gfCNCPoint2[13248] = {X 390.9830, Y 62.2246, Z -3.0000, A 0.000, B 0.000, C 0.000 }
gfCNCPoint2[13249] = {X 390.3072, Y 62.7207, Z -3.0000, A 0.000, B 0.000, C 0.000 }
gfCNCPoint2[13250] = {X 389.5499, Y 63.0803, Z -3.0000, A 0.000, B 0.000, C 0.000 }
gfCNCPoint2[13251] = {X 388.7383, Y 63.2905, Z -3.0000, A 0.000, B 0.000, C 0.000 }
gfCNCPoint2[13252] = {X 388.7383, Y 83.9247, Z -3.0000, A 0.000, B 0.000, C 0.000 }
gfCNCPoint2[13253] = {X 388.7363, Y 84.6149, Z -3.0000, A 0.000, B 0.000, C 0.000 }
gfCNCPoint2[13254] = {X 388.6762, Y 86.2799, Z -3.0000, A 0.000, B 0.000, C 0.000 }
gfCNCPoint2[13255] = {X 388.4710, Y 87.9334, Z -3.0000, A 0.000, B 0.000, C 0.000 }
gfCNCPoint2[13256] = {X 388.1223, Y 89.5626, Z -3.0000, A 0.000, B 0.000, C 0.000 }
gfCNCPoint2[13257] = {X 387.5865, Y 91.1607, Z -3.0000, A 0.000, B 0.000, C 0.000 }
gfCNCPoint2[13258] = {X 386.8319, Y 92.6679, Z -3.0000, A 0.000, B 0.000, C 0.000 }
gfCNCPoint2[13259] = {X 385.8732, Y 94.0543, Z -3.0000, A 0.000, B 0.000, C 0.000 }
gfCNCPoint2[13260] = {X 384.7295, Y 95.2924, Z -3.0000, A 0.000, B 0.000, C 0.000 }
gfCNCPoint2[13261] = {X 383.5014, Y 96.3480, Z -3.0000, A 0.000, B 0.000, C 0.000 }
gfCNCPoint2[13262] = {X 382.1865, Y 97.2935, Z -3.0000, A 0.000, B 0.000, C 0.000 }
gfCNCPoint2[13263] = {X 382.4496, Y 97.6950, Z -3.0000, A 0.000, B 0.000, C 0.000 }
gfCNCPoint2[13264] = {X 391.5259, Y 97.6950, Z -3.0000, A 0.000, B 0.000, C 0.000 }
gfCNCPoint2[13265] = {X 391.5259, Y 97.0659, Z -3.0000, A 0.000, B 0.000, C 0.000 }
gfCNCPoint2[13266] = {X 391.6192, Y 96.1166, Z -3.0000, A 0.000, B 0.000, C 0.000 }
gfCNCPoint2[13267] = {X 391.8953, Y 95.2035, Z -3.0000, A 0.000, B 0.000, C 0.000 }
gfCNCPoint2[13268] = {X 392.3439, Y 94.3615, Z -3.0000, A 0.000, B 0.000, C 0.000 }
gfCNCPoint2[13269] = {X 392.9476, Y 93.6229, Z -3.0000, A 0.000, B 0.000, C 0.000 }
gfCNCPoint2[13270] = {X 393.6835, Y 93.0159, Z -3.0000, A 0.000, B 0.000, C 0.000 }
gfCNCPoint2[13271] = {X 394.5234, Y 92.5637, Z -3.0000, A 0.000, B 0.000, C 0.000 }
gfCNCPoint2[13272] = {X 395.4353, Y 92.2834, Z -3.0000, A 0.000, B 0.000, C 0.000 }
gfCNCPoint2[13273] = {X 396.3843, Y 92.1860, Z -3.0000, A 0.000, B 0.000, C 0.000 }
gfCNCPoint2[13274] = {X 397.3061, Y 92.1465, Z -3.0000, A 0.000, B 0.000, C 0.000 }
gfCNCPoint2[13275] = {X 398.2246, Y 92.0592, Z -3.0000, A 0.000, B 0.000, C 0.000 }
gfCNCPoint2[13276] = {X 398.7527, Y 91.9311, Z -3.0000, A 0.000, B 0.000, C 0.000 }
gfCNCPoint2[13277] = {X 399.2389, Y 91.6885, Z -3.0000, A 0.000, B 0.000, C 0.000 }
gfCNCPoint2[13278] = {X 426.8276, Y 74.0193, Z -3.0000, A 0.000, B 0.000, C 0.000 }
gfCNCPoint2[13279] = {X 403.5508, Y 64.8864, Z -3.0000, A 0.000, B 0.000, C 0.000 }
gfCNCPoint2[13280] = {X 401.9168, Y 64.3451, Z -3.0000, A 0.000, B 0.000, C 0.000 }
gfCNCPoint2[13281] = {X 400.2332, Y 63.9861, Z -3.0000, A 0.000, B 0.000, C 0.000 }
gfCNCPoint2[13282] = {X 398.5205, Y 63.8139, Z -3.0000, A 0.000, B 0.000, C 0.000 }
gfCNCPoint2[13283] = {X 397.5547, Y 63.7099, Z -3.0000, A 0.000, B 0.000, C 0.000 }
gfCNCPoint2[13284] = {X 396.6287, Y 63.4166, Z -3.0000, A 0.000, B 0.000, C 0.000 }
gfCNCPoint2[13285] = {X 395.7791, Y 62.9458, Z -3.0000, A 0.000, B 0.000, C 0.000 }
gfCNCPoint2[13286] = {X 395.0396, Y 62.3160, Z -3.0000, A 0.000, B 0.000, C 0.000 }
gfCNCPoint2[13287] = {X 394.4659, Y 61.5933, Z -3.0000, A 0.000, B 0.000, C 0.000 }
gfCNCPoint2[13288] = {X 394.0385, Y 60.7756, Z -3.0000, A 0.000, B 0.000, C 0.000 }
gfCNCPoint2[13289] = {X 393.7727, Y 59.8921, Z -3.0000, A 0.000, B 0.000, C 0.000 }
gfCNCPoint2[13290] = {X 393.6779, Y 58.9744, Z -3.0000, A 0.000, B 0.000, C 0.000 }
gfCNCPoint2[13291] = {X 393.6777, Y 58.0000, Z -3.0000, A 0.000, B 0.000, C 0.000 }
gfCNCPoint2[13292] = {X 393.7668, Y 57.0718, Z -3.0000, A 0.000, B 0.000, C 0.000 }
gfCNCPoint2[13293] = {X 394.0309, Y 56.1774, Z -3.0000, A 0.000, B 0.000, C 0.000 }
gfCNCPoint2[13294] = {X 394.4602, Y 55.3496, Z -3.0000, A 0.000, B 0.000, C 0.000 }
gfCNCPoint2[13295] = {X 395.0391, Y 54.6186, Z -3.0000, A 0.000, B 0.000, C 0.000 }
gfCNCPoint2[13296] = {X 395.7864, Y 53.9833, Z -3.0000, A 0.000, B 0.000, C 0.000 }
gfCNCPoint2[13297] = {X 396.6455, Y 53.5102, Z -3.0000, A 0.000, B 0.000, C 0.000 }
gfCNCPoint2[13298] = {X 397.5819, Y 53.2186, Z -3.0000, A 0.000, B 0.000, C 0.000 }
gfCNCPoint2[13299] = {X 398.5577, Y 53.1200, Z -3.0000, A 0.000, B 0.000, C 0.000 }
gfCNCPoint2[13300] = {X 419.4886, Y 53.1200, Z -3.0000, A 0.000, B 0.000, C 0.000 }
gfCNCPoint2[13301] = {X 420.5534, Y 53.2376, Z -3.0000, A 0.000, B 0.000, C 0.000 }
gfCNCPoint2[13302] = {X 421.5670, Y 53.5847, Z -3.0000, A 0.000, B 0.000, C 0.000 }
gfCNCPoint2[13303] = {X 422.4803, Y 54.1446, Z -3.0000, A 0.000, B 0.000, C 0.000 }
gfCNCPoint2[13304] = {X 423.2495, Y 54.8903, Z -3.0000, A 0.000, B 0.000, C 0.000 }
gfCNCPoint2[13305] = {X 423.8374, Y 55.7859, Z -3.0000, A 0.000, B 0.000, C 0.000 }
gfCNCPoint2[13306] = {X 424.2157, Y 56.7881, Z -3.0000, A 0.000, B 0.000, C 0.000 }
gfCNCPoint2[13307] = {X 424.3663, Y 57.8488, Z -3.0000, A 0.000, B 0.000, C 0.000 }
gfCNCPoint2[13308] = {X 429.8190, Y 59.9739, Z -3.0000, A 0.000, B 0.000, C 0.000 }
gfCNCPoint2[13309] = {X 457.3006, Y 70.8772, Z -3.0000, A 0.000, B 0.000, C 0.000 }
gfCNCPoint2[13310] = {X 457.2996, Y 63.6742, Z -3.0000, A 0.000, B 0.000, C 0.000 }
gfCNCPoint2[13311] = {X 456.2913, Y 63.3059, Z -3.0000, A 0.000, B 0.000, C 0.000 }
gfCNCPoint2[13312] = {X 455.3879, Y 62.7260, Z -3.0000, A 0.000, B 0.000, C 0.000 }
gfCNCPoint2[13313] = {X 454.6331, Y 61.9627, Z -3.0000, A 0.000, B 0.000, C 0.000 }
gfCNCPoint2[13314] = {X 454.0635, Y 61.0528, Z -3.0000, A 0.000, B 0.000, C 0.000 }
gfCNCPoint2[13315] = {X 453.7067, Y 60.0403, Z -3.0000, A 0.000, B 0.000, C 0.000 }
gfCNCPoint2[13316] = {X 453.5798, Y 58.9744, Z -3.0000, A 0.000, B 0.000, C 0.000 }
gfCNCPoint2[13317] = {X 453.5796, Y 58.0000, Z -3.0000, A 0.000, B 0.000, C 0.000 }
gfCNCPoint2[13318] = {X 453.6734, Y 57.0480, Z -3.0000, A 0.000, B 0.000, C 0.000 }
gfCNCPoint2[13319] = {X 453.9511, Y 56.1325, Z -3.0000, A 0.000, B 0.000, C 0.000 }
gfCNCPoint2[13320] = {X 454.4020, Y 55.2888, Z -3.0000, A 0.000, B 0.000, C 0.000 }
gfCNCPoint2[13321] = {X 455.0089, Y 54.5493, Z -3.0000, A 0.000, B 0.000, C 0.000 }
gfCNCPoint2[13322] = {X 455.7484, Y 53.9424, Z -3.0000, A 0.000, B 0.000, C 0.000 }
gfCNCPoint2[13323] = {X 456.5921, Y 53.4915, Z -3.0000, A 0.000, B 0.000, C 0.000 }
gfCNCPoint2[13324] = {X 457.5076, Y 53.2138, Z -3.0000, A 0.000, B 0.000, C 0.000 }
gfCNCPoint2[13325] = {X 458.4596, Y 53.1200, Z -3.0000, A 0.000, B 0.000, C 0.000 }
gfCNCPoint2[13326] = {X 475.0000, Y 53.1200, Z -3.0000, A 0.000, B 0.000, C 0.000 }
gfCNCPoint2[13327] = {X 475.9520, Y 53.2138, Z -3.0000, A 0.000, B 0.000, C 0.000 }
gfCNCPoint2[13328] = {X 476.8675, Y 53.4915, Z -3.0000, A 0.000, B 0.000, C 0.000 }
gfCNCPoint2[13329] = {X 477.7112, Y 53.9424, Z -3.0000, A 0.000, B 0.000, C 0.000 }
gfCNCPoint2[13330] = {X 478.4507, Y 54.5493, Z -3.0000, A 0.000, B 0.000, C 0.000 }
gfCNCPoint2[13331] = {X 479.0576, Y 55.2888, Z -3.0000, A 0.000, B 0.000, C 0.000 }
gfCNCPoint2[13332] = {X 479.5085, Y 56.1325, Z -3.0000, A 0.000, B 0.000, C 0.000 }
gfCNCPoint2[13333] = {X 479.7862, Y 57.0480, Z -3.0000, A 0.000, B 0.000, C 0.000 }
gfCNCPoint2[13334] = {X 479.8800, Y 58.0000, Z -3.0000, A 0.000, B 0.000, C 0.000 }
gfCNCPoint2[13335] = {X 479.8798, Y 58.9744, Z -3.0000, A 0.000, B 0.000, C 0.000 }
gfCNCPoint2[13336] = {X 479.7529, Y 60.0404, Z -3.0000, A 0.000, B 0.000, C 0.000 }
gfCNCPoint2[13337] = {X 479.3960, Y 61.0529, Z -3.0000, A 0.000, B 0.000, C 0.000 }
gfCNCPoint2[13338] = {X 478.8264, Y 61.9628, Z -3.0000, A 0.000, B 0.000, C 0.000 }
gfCNCPoint2[13339] = {X 478.0716, Y 62.7261, Z -3.0000, A 0.000, B 0.000, C 0.000 }
gfCNCPoint2[13340] = {X 477.1681, Y 63.3060, Z -3.0000, A 0.000, B 0.000, C 0.000 }
gfCNCPoint2[13341] = {X 476.1597, Y 63.6743, Z -3.0000, A 0.000, B 0.000, C 0.000 }
gfCNCPoint2[13342] = {X 476.1601, Y 92.3320, Z -3.0000, A 0.000, B 0.000, C 0.000 }
gfCNCPoint2[13343] = {X 476.3629, Y 92.3914, Z -3.0000, A 0.000, B 0.000, C 0.000 }
gfCNCPoint2[13344] = {X 476.5640, Y 92.4558, Z -3.0000, A 0.000, B 0.000, C 0.000 }
gfCNCPoint2[13345] = {X 477.4819, Y 92.8728, Z -3.0000, A 0.000, B 0.000, C 0.000 }
gfCNCPoint2[13346] = {X 478.2938, Y 93.4704, Z -3.0000, A 0.000, B 0.000, C 0.000 }
gfCNCPoint2[13347] = {X 478.9647, Y 94.2227, Z -3.0000, A 0.000, B 0.000, C 0.000 }
gfCNCPoint2[13348] = {X 479.4658, Y 95.0975, Z -3.0000, A 0.000, B 0.000, C 0.000 }
gfCNCPoint2[13349] = {X 479.7753, Y 96.0569, Z -3.0000, A 0.000, B 0.000, C 0.000 }
gfCNCPoint2[13350] = {X 479.8800, Y 97.0595, Z -3.0000, A 0.000, B 0.000, C 0.000 }
gfCNCPoint2[13351] = {X 479.8800, Y 97.6950, Z -3.0000, A 0.000, B 0.000, C 0.000 }
gfCNCPoint2[13352] = {X 479.4000, Y 97.6950, Z -3.0000, A 0.000, B 0.000, C 0.000 }
gfCNCPoint2[13353] = {X 479.4000, Y 98.0000, Z -3.0000, A 0.000, B 0.000, C 0.000 }
gfCNCPoint2[13354] = {X 479.2897, Y 98.9791, Z -3.0000, A 0.000, B 0.000, C 0.000 }
gfCNCPoint2[13355] = {X 478.9643, Y 99.9091, Z -3.0000, A 0.000, B 0.000, C 0.000 }
gfCNCPoint2[13356] = {X 478.4401, Y 100.7434, Z -3.0000, A 0.000, B 0.000, C 0.000 }
gfCNCPoint2[13357] = {X 477.7434, Y 101.4401, Z -3.0000, A 0.000, B 0.000, C 0.000 }
gfCNCPoint2[13358] = {X 476.9091, Y 101.9643, Z -3.0000, A 0.000, B 0.000, C 0.000 }
gfCNCPoint2[13359] = {X 475.9791, Y 102.2897, Z -3.0000, A 0.000, B 0.000, C 0.000 }
gfCNCPoint2[13360] = {X 475.0000, Y 102.4000, Z -3.0000, A 0.000, B 0.000, C 0.000 }
gfCNCPoint2[13361] = {X 458.4596, Y 102.4000, Z -3.0000, A 0.000, B 0.000, C 0.000 }
gfCNCPoint2[13362] = {X 457.4805, Y 102.2897, Z -3.0000, A 0.000, B 0.000, C 0.000 }
gfCNCPoint2[13363] = {X 456.5505, Y 101.9643, Z -3.0000, A 0.000, B 0.000, C 0.000 }
gfCNCPoint2[13364] = {X 455.7162, Y 101.4401, Z -3.0000, A 0.000, B 0.000, C 0.000 }
gfCNCPoint2[13365] = {X 455.0195, Y 100.7434, Z -3.0000, A 0.000, B 0.000, C 0.000 }
gfCNCPoint2[13366] = {X 454.4953, Y 99.9091, Z -3.0000, A 0.000, B 0.000, C 0.000 }
gfCNCPoint2[13367] = {X 454.1699, Y 98.9791, Z -3.0000, A 0.000, B 0.000, C 0.000 }
gfCNCPoint2[13368] = {X 454.0596, Y 98.0000, Z -3.0000, A 0.000, B 0.000, C 0.000 }
gfCNCPoint2[13369] = {X 454.0596, Y 97.0659, Z -3.0000, A 0.000, B 0.000, C 0.000 }
gfCNCPoint2[13370] = {X 454.1492, Y 96.1826, Z -3.0000, A 0.000, B 0.000, C 0.000 }
gfCNCPoint2[13371] = {X 454.4143, Y 95.3353, Z -3.0000, A 0.000, B 0.000, C 0.000 }
gfCNCPoint2[13372] = {X 454.8440, Y 94.5584, Z -3.0000, A 0.000, B 0.000, C 0.000 }
gfCNCPoint2[13373] = {X 455.4210, Y 93.8836, Z -3.0000, A 0.000, B 0.000, C 0.000 }
gfCNCPoint2[13374] = {X 456.1217, Y 93.3384, Z -3.0000, A 0.000, B 0.000, C 0.000 }
gfCNCPoint2[13375] = {X 456.9176, Y 92.9450, Z -3.0000, A 0.000, B 0.000, C 0.000 }
gfCNCPoint2[13376] = {X 457.7763, Y 92.7193, Z -3.0000, A 0.000, B 0.000, C 0.000 }
gfCNCPoint2[13377] = {X 457.7763, Y 85.6495, Z -3.0000, A 0.000, B 0.000, C 0.000 }
gfCNCPoint2[13378] = {X 444.8675, Y 80.5893, Z -3.0000, A 0.000, B 0.000, C 0.000 }
gfCNCPoint2[13379] = {X 420.1033, Y 96.6314, Z -3.0000, A 0.000, B 0.000, C 0.000 }
gfCNCPoint2[13380] = {X 420.1067, Y 97.0659, Z -3.0000, A 0.000, B 0.000, C 0.000 }
gfCNCPoint2[13381] = {X 420.1067, Y 98.0000, Z -3.0000, A 0.000, B 0.000, C 0.000 }
gfCNCPoint2[13382] = {X 419.9964, Y 98.9791, Z -3.0000, A 0.000, B 0.000, C 0.000 }
gfCNCPoint2[13383] = {X 419.6710, Y 99.9091, Z -3.0000, A 0.000, B 0.000, C 0.000 }
gfCNCPoint2[13384] = {X 419.1468, Y 100.7434, Z -3.0000, A 0.000, B 0.000, C 0.000 }
gfCNCPoint2[13385] = {X 418.4501, Y 101.4401, Z -3.0000, A 0.000, B 0.000, C 0.000 }
gfCNCPoint2[13386] = {X 417.6158, Y 101.9643, Z -3.0000, A 0.000, B 0.000, C 0.000 }
gfCNCPoint2[13387] = {X 416.6858, Y 102.2897, Z -3.0000, A 0.000, B 0.000, C 0.000 }
gfCNCPoint2[13388] = {X 415.7067, Y 102.4000, Z -3.0000, A 0.000, B 0.000, C 0.000 }
gfCNCPoint2[13389] = {X 396.4059, Y 102.4000, Z -3.0000, A 0.000, B 0.000, C 0.000 }
gfCNCPoint2[13390] = {X 395.4269, Y 102.2897, Z -3.0000, A 0.000, B 0.000, C 0.000 }
gfCNCPoint2[13391] = {X 394.4969, Y 101.9643, Z -3.0000, A 0.000, B 0.000, C 0.000 }
gfCNCPoint2[13392] = {X 393.6626, Y 101.4401, Z -3.0000, A 0.000, B 0.000, C 0.000 }
gfCNCPoint2[13393] = {X 392.9659, Y 100.7434, Z -3.0000, A 0.000, B 0.000, C 0.000 }
gfCNCPoint2[13394] = {X 392.4417, Y 99.9091, Z -3.0000, A 0.000, B 0.000, C 0.000 }
gfCNCPoint2[13395] = {X 392.1163, Y 98.9791, Z -3.0000, A 0.000, B 0.000, C 0.000 }
gfCNCPoint2[13396] = {X 392.0059, Y 98.0000, Z -3.0000, A 0.000, B 0.000, C 0.000 }
gfCNCPoint2[13397] = {X 392.0059, Y 97.0659, Z -3.0000, A 0.000, B 0.000, C 0.000 }
gfCNCPoint2[13398] = {X 392.1157, Y 96.0892, Z -3.0000, A 0.000, B 0.000, C 0.000 }
gfCNCPoint2[13399] = {X 392.4396, Y 95.1611, Z -3.0000, A 0.000, B 0.000, C 0.000 }
gfCNCPoint2[13400] = {X 392.9614, Y 94.3282, Z -3.0000, A 0.000, B 0.000, C 0.000 }
gfCNCPoint2[13401] = {X 393.6552, Y 93.6318, Z -3.0000, A 0.000, B 0.000, C 0.000 }
gfCNCPoint2[13402] = {X 394.4861, Y 93.1068, Z -3.0000, A 0.000, B 0.000, C 0.000 }
gfCNCPoint2[13403] = {X 395.4129, Y 92.7795, Z -3.0000, A 0.000, B 0.000, C 0.000 }
gfCNCPoint2[13404] = {X 396.3893, Y 92.6660, Z -3.0000, A 0.000, B 0.000, C 0.000 }
gfCNCPoint2[13405] = {X 397.3382, Y 92.6254, Z -3.0000, A 0.000, B 0.000, C 0.000 }
gfCNCPoint2[13406] = {X 398.2836, Y 92.5356, Z -3.0000, A 0.000, B 0.000, C 0.000 }
gfCNCPoint2[13407] = {X 398.9175, Y 92.3819, Z -3.0000, A 0.000, B 0.000, C 0.000 }
gfCNCPoint2[13408] = {X 399.5010, Y 92.0906, Z -3.0000, A 0.000, B 0.000, C 0.000 }
gfCNCPoint2[13409] = {X 405.1774, Y 88.4328, Z -3.0000, A 0.000, B 0.000, C 0.000 }
gfCNCPoint2[13410] = {X 427.8795, Y 73.9165, Z -3.0000, A 0.000, B 0.000, C 0.000 }
gfCNCPoint2[13411] = {X 403.7262, Y 64.4396, Z -3.0000, A 0.000, B 0.000, C 0.000 }
gfCNCPoint2[13412] = {X 402.0392, Y 63.8810, Z -3.0000, A 0.000, B 0.000, C 0.000 }
gfCNCPoint2[13413] = {X 400.3011, Y 63.5109, Z -3.0000, A 0.000, B 0.000, C 0.000 }
gfCNCPoint2[13414] = {X 398.5329, Y 63.3340, Z -3.0000, A 0.000, B 0.000, C 0.000 }
gfCNCPoint2[13415] = {X 397.5579, Y 63.2190, Z -3.0000, A 0.000, B 0.000, C 0.000 }
gfCNCPoint2[13416] = {X 396.6327, Y 62.8906, Z -3.0000, A 0.000, B 0.000, C 0.000 }
gfCNCPoint2[13417] = {X 395.8033, Y 62.3652, Z -3.0000, A 0.000, B 0.000, C 0.000 }
gfCNCPoint2[13418] = {X 395.1110, Y 61.6691, Z -3.0000, A 0.000, B 0.000, C 0.000 }
gfCNCPoint2[13419] = {X 394.5904, Y 60.8367, Z -3.0000, A 0.000, B 0.000, C 0.000 }
gfCNCPoint2[13420] = {X 394.2672, Y 59.9097, Z -3.0000, A 0.000, B 0.000, C 0.000 }
gfCNCPoint2[13421] = {X 394.1577, Y 58.9340, Z -3.0000, A 0.000, B 0.000, C 0.000 }
gfCNCPoint2[13422] = {X 394.1577, Y 58.0000, Z -3.0000, A 0.000, B 0.000, C 0.000 }
gfCNCPoint2[13423] = {X 394.2680, Y 57.0209, Z -3.0000, A 0.000, B 0.000, C 0.000 }
gfCNCPoint2[13424] = {X 394.5935, Y 56.0909, Z -3.0000, A 0.000, B 0.000, C 0.000 }
gfCNCPoint2[13425] = {X 395.1177, Y 55.2566, Z -3.0000, A 0.000, B 0.000, C 0.000 }
gfCNCPoint2[13426] = {X 395.8144, Y 54.5599, Z -3.0000, A 0.000, B 0.000, C 0.000 }
gfCNCPoint2[13427] = {X 396.6486, Y 54.0357, Z -3.0000, A 0.000, B 0.000, C 0.000 }
gfCNCPoint2[13428] = {X 397.5786, Y 53.7103, Z -3.0000, A 0.000, B 0.000, C 0.000 }
gfCNCPoint2[13429] = {X 398.5577, Y 53.6000, Z -3.0000, A 0.000, B 0.000, C 0.000 }
gfCNCPoint2[13430] = {X 419.4886, Y 53.6000, Z -3.0000, A 0.000, B 0.000, C 0.000 }
gfCNCPoint2[13431] = {X 420.4677, Y 53.7103, Z -3.0000, A 0.000, B 0.000, C 0.000 }
gfCNCPoint2[13432] = {X 421.3977, Y 54.0357, Z -3.0000, A 0.000, B 0.000, C 0.000 }
gfCNCPoint2[13433] = {X 422.2320, Y 54.5599, Z -3.0000, A 0.000, B 0.000, C 0.000 }
gfCNCPoint2[13434] = {X 422.9287, Y 55.2566, Z -3.0000, A 0.000, B 0.000, C 0.000 }
gfCNCPoint2[13435] = {X 423.4529, Y 56.0909, Z -3.0000, A 0.000, B 0.000, C 0.000 }
gfCNCPoint2[13436] = {X 423.7783, Y 57.0209, Z -3.0000, A 0.000, B 0.000, C 0.000 }
gfCNCPoint2[13437] = {X 423.8886, Y 58.0000, Z -3.0000, A 0.000, B 0.000, C 0.000 }
gfCNCPoint2[13438] = {X 423.8886, Y 58.1778, Z -3.0000, A 0.000, B 0.000, C 0.000 }
gfCNCPoint2[13439] = {X 429.6420, Y 60.4200, Z -3.0000, A 0.000, B 0.000, C 0.000 }
gfCNCPoint2[13440] = {X 457.7807, Y 71.5841, Z -3.0000, A 0.000, B 0.000, C 0.000 }
gfCNCPoint2[13441] = {X 457.7796, Y 63.2812, Z -3.0000, A 0.000, B 0.000, C 0.000 }
gfCNCPoint2[13442] = {X 456.9203, Y 63.0560, Z -3.0000, A 0.000, B 0.000, C 0.000 }
gfCNCPoint2[13443] = {X 456.1237, Y 62.6628, Z -3.0000, A 0.000, B 0.000, C 0.000 }
gfCNCPoint2[13444] = {X 455.4224, Y 62.1177, Z -3.0000, A 0.000, B 0.000, C 0.000 }
gfCNCPoint2[13445] = {X 454.8448, Y 61.4427, Z -3.0000, A 0.000, B 0.000, C 0.000 }
gfCNCPoint2[13446] = {X 454.4146, Y 60.6656, Z -3.0000, A 0.000, B 0.000, C 0.000 }
gfCNCPoint2[13447] = {X 454.1493, Y 59.8178, Z -3.0000, A 0.000, B 0.000, C 0.000 }
gfCNCPoint2[13448] = {X 454.0596, Y 58.9340, Z -3.0000, A 0.000, B 0.000, C 0.000 }
gfCNCPoint2[13449] = {X 454.0596, Y 58.0000, Z -3.0000, A 0.000, B 0.000, C 0.000 }
gfCNCPoint2[13450] = {X 454.1699, Y 57.0209, Z -3.0000, A 0.000, B 0.000, C 0.000 }
gfCNCPoint2[13451] = {X 454.4953, Y 56.0909, Z -3.0000, A 0.000, B 0.000, C 0.000 }
gfCNCPoint2[13452] = {X 455.0195, Y 55.2566, Z -3.0000, A 0.000, B 0.000, C 0.000 }
gfCNCPoint2[13453] = {X 455.7162, Y 54.5599, Z -3.0000, A 0.000, B 0.000, C 0.000 }
gfCNCPoint2[13454] = {X 456.5505, Y 54.0357, Z -3.0000, A 0.000, B 0.000, C 0.000 }
gfCNCPoint2[13455] = {X 457.4805, Y 53.7103, Z -3.0000, A 0.000, B 0.000, C 0.000 }
gfCNCPoint2[13456] = {X 458.4596, Y 53.6000, Z -3.0000, A 0.000, B 0.000, C 0.000 }
gfCNCPoint2[13457] = {X 475.0000, Y 53.6000, Z -3.0000, A 0.000, B 0.000, C 0.000 }
gfCNCPoint2[13458] = {X 475.9791, Y 53.7103, Z -3.0000, A 0.000, B 0.000, C 0.000 }
gfCNCPoint2[13459] = {X 476.9091, Y 54.0357, Z -3.0000, A 0.000, B 0.000, C 0.000 }
gfCNCPoint2[13460] = {X 477.7434, Y 54.5599, Z -3.0000, A 0.000, B 0.000, C 0.000 }
gfCNCPoint2[13461] = {X 478.4401, Y 55.2566, Z -3.0000, A 0.000, B 0.000, C 0.000 }
gfCNCPoint2[13462] = {X 478.9643, Y 56.0909, Z -3.0000, A 0.000, B 0.000, C 0.000 }
gfCNCPoint2[13463] = {X 479.2897, Y 57.0209, Z -3.0000, A 0.000, B 0.000, C 0.000 }
gfCNCPoint2[13464] = {X 479.4000, Y 58.0000, Z -3.0000, A 0.000, B 0.000, C 0.000 }
gfCNCPoint2[13465] = {X 479.3998, Y 58.9704, Z -3.0000, A 0.000, B 0.000, C 0.000 }
gfCNCPoint2[13466] = {X 479.3040, Y 59.8484, Z -3.0000, A 0.000, B 0.000, C 0.000 }
gfCNCPoint2[13467] = {X 479.0347, Y 60.6895, Z -3.0000, A 0.000, B 0.000, C 0.000 }
gfCNCPoint2[13468] = {X 478.6028, Y 61.4599, Z -3.0000, A 0.000, B 0.000, C 0.000 }
gfCNCPoint2[13469] = {X 478.0258, Y 62.1285, Z -3.0000, A 0.000, B 0.000, C 0.000 }
gfCNCPoint2[13470] = {X 477.3269, Y 62.6685, Z -3.0000, A 0.000, B 0.000, C 0.000 }
gfCNCPoint2[13471] = {X 476.5342, Y 63.0579, Z -3.0000, A 0.000, B 0.000, C 0.000 }
gfCNCPoint2[13472] = {X 475.6797, Y 63.2812, Z -3.0000, A 0.000, B 0.000, C 0.000 }
gfCNCPoint2[13473] = {X 475.6801, Y 92.7047, Z -3.0000, A 0.000, B 0.000, C 0.000 }
gfCNCPoint2[13474] = {X 476.0485, Y 92.7992, Z -3.0000, A 0.000, B 0.000, C 0.000 }
gfCNCPoint2[13475] = {X 476.4120, Y 92.9111, Z -3.0000, A 0.000, B 0.000, C 0.000 }
gfCNCPoint2[13476] = {X 477.2390, Y 93.2868, Z -3.0000, A 0.000, B 0.000, C 0.000 }
gfCNCPoint2[13477] = {X 477.9706, Y 93.8253, Z -3.0000, A 0.000, B 0.000, C 0.000 }
gfCNCPoint2[13478] = {X 478.5752, Y 94.5033, Z -3.0000, A 0.000, B 0.000, C 0.000 }
gfCNCPoint2[13479] = {X 479.0267, Y 95.2915, Z -3.0000, A 0.000, B 0.000, C 0.000 }
gfCNCPoint2[13480] = {X 479.3057, Y 96.1561, Z -3.0000, A 0.000, B 0.000, C 0.000 }
gfCNCPoint2[13481] = {X 479.4000, Y 97.0595, Z -3.0000, A 0.000, B 0.000, C 0.000 }
gfCNCPoint2[13482] = {X 479.4000, Y 97.6950, Z -3.0000, A 0.000, B 0.000, C 0.000 }
gfCNCPoint2[13483] = {X 479.8800, Y 97.6950, Z -3.0000, A 0.000, B 0.000, C 0.000 }
gfCNCPoint2[13484] = {X 507.6818, Y 97.6950, Z -3.0000, A 0.000, B 0.000, C 0.000 }
gfCNCPoint2[13485] = {X 507.6818, Y 100.0950, Z -3.0000, A 0.000, B 0.000, C 0.000 }
gfCNCPoint2[13486] = {X 600.0148, Y 100.0950, Z -3.0000, A 0.000, B 0.000, C 0.000 }
gfCNCPoint2[13487] = {X 600.0672, Y 100.0698, Z -3.0000, A 0.000, B 0.000, C 0.000 }
gfCNCPoint2[13488] = {X 600.0948, Y 100.0187, Z -3.0000, A 0.000, B 0.000, C 0.000 }
gfCNCPoint2[13489] = {X 600.0965, Y 99.1431, Z -3.0000, A 0.000, B 0.000, C 0.000 }
gfCNCPoint2[13490] = {X 600.0965, Y 49.8790, Z -3.0000, A 0.000, B 0.000, C 0.000 }
gfCNCPoint2[13491] = {X 601.1111, Y 49.7518, Z -3.0000, A 0.000, B 0.000, C 0.000 }
gfCNCPoint2[13492] = {X 602.0769, Y 49.4160, Z -3.0000, A 0.000, B 0.000, C 0.000 }
gfCNCPoint2[13493] = {X 602.9515, Y 48.8863, Z -3.0000, A 0.000, B 0.000, C 0.000 }
gfCNCPoint2[13494] = {X 603.6965, Y 48.1859, Z -3.0000, A 0.000, B 0.000, C 0.000 }
gfCNCPoint2[13495] = {X 603.6965, Y 47.3866, Z -3.0000, A 0.000, B 0.000, C 0.000 }
gfCNCPoint2[13496] = {X 603.1502, Y 48.0718, Z -3.0000, A 0.000, B 0.000, C 0.000 }
gfCNCPoint2[13497] = {X 602.4790, Y 48.6352, Z -3.0000, A 0.000, B 0.000, C 0.000 }
gfCNCPoint2[13498] = {X 601.7094, Y 49.0544, Z -3.0000, A 0.000, B 0.000, C 0.000 }
gfCNCPoint2[13499] = {X 600.8720, Y 49.3127, Z -3.0000, A 0.000, B 0.000, C 0.000 }
gfCNCPoint2[13500] = {X 600.0000, Y 49.4000, Z -3.0000, A 0.000, B 0.000, C 0.000 }
gfCNCPoint2[13501] = {X 593.5565, Y 49.4000, Z -3.0000, A 0.000, B 0.000, C 0.000 }
gfCNCPoint2[13502] = {X 592.5988, Y 49.2945, Z -3.0000, A 0.000, B 0.000, C 0.000 }
gfCNCPoint2[13503] = {X 591.6870, Y 48.9831, Z -3.0000, A 0.000, B 0.000, C 0.000 }
gfCNCPoint2[13504] = {X 590.8648, Y 48.4806, Z -3.0000, A 0.000, B 0.000, C 0.000 }
gfCNCPoint2[13505] = {X 590.1717, Y 47.8112, Z -3.0000, A 0.000, B 0.000, C 0.000 }
gfCNCPoint2[13506] = {X 589.6410, Y 47.0071, Z -3.0000, A 0.000, B 0.000, C 0.000 }
gfCNCPoint2[13507] = {X 589.3741, Y 46.3664, Z -3.0000, A 0.000, B 0.000, C 0.000 }
gfCNCPoint2[13508] = {X 589.2113, Y 45.6918, Z -3.0000, A 0.000, B 0.000, C 0.000 }
gfCNCPoint2[13509] = {X 589.1565, Y 45.0000, Z -3.0000, A 0.000, B 0.000, C 0.000 }
gfCNCPoint2[13510] = {X 589.1565, Y 44.0640, Z -3.0000, A 0.000, B 0.000, C 0.000 }
gfCNCPoint2[13511] = {X 589.2611, Y 43.1277, Z -3.0000, A 0.000, B 0.000, C 0.000 }
gfCNCPoint2[13512] = {X 589.5608, Y 42.2345, Z -3.0000, A 0.000, B 0.000, C 0.000 }
gfCNCPoint2[13513] = {X 590.0421, Y 41.4246, Z -3.0000, A 0.000, B 0.000, C 0.000 }
gfCNCPoint2[13514] = {X 590.6833, Y 40.7344, Z -3.0000, A 0.000, B 0.000, C 0.000 }
gfCNCPoint2[13515] = {X 590.6848, Y 40.3069, Z -3.0000, A 0.000, B 0.000, C 0.000 }
gfCNCPoint2[13516] = {X 590.6836, Y 33.9394, Z -3.0000, A 0.000, B 0.000, C 0.000 }
gfCNCPoint2[13517] = {X 585.5192, Y 46.6830, Z -3.0000, A 0.000, B 0.000, C 0.000 }
gfCNCPoint2[13518] = {X 585.4476, Y 46.8466, Z -3.0000, A 0.000, B 0.000, C 0.000 }
gfCNCPoint2[13519] = {X 585.3694, Y 47.0071, Z -3.0000, A 0.000, B 0.000, C 0.000 }
gfCNCPoint2[13520] = {X 584.8417, Y 47.8075, Z -3.0000, A 0.000, B 0.000, C 0.000 }
gfCNCPoint2[13521] = {X 584.1532, Y 48.4747, Z -3.0000, A 0.000, B 0.000, C 0.000 }
gfCNCPoint2[13522] = {X 583.3365, Y 48.9769, Z -3.0000, A 0.000, B 0.000, C 0.000 }
gfCNCPoint2[13523] = {X 582.4111, Y 49.2946, Z -3.0000, A 0.000, B 0.000, C 0.000 }
gfCNCPoint2[13524] = {X 581.4384, Y 49.4000, Z -3.0000, A 0.000, B 0.000, C 0.000 }
gfCNCPoint2[13525] = {X 580.4664, Y 49.2878, Z -3.0000, A 0.000, B 0.000, C 0.000 }
gfCNCPoint2[13526] = {X 579.5433, Y 48.9635, Z -3.0000, A 0.000, B 0.000, C 0.000 }
gfCNCPoint2[13527] = {X 578.7146, Y 48.4433, Z -3.0000, A 0.000, B 0.000, C 0.000 }
gfCNCPoint2[13528] = {X 578.0214, Y 47.7529, Z -3.0000, A 0.000, B 0.000, C 0.000 }
gfCNCPoint2[13529] = {X 577.4979, Y 46.9263, Z -3.0000, A 0.000, B 0.000, C 0.000 }
gfCNCPoint2[13530] = {X 577.4375, Y 46.7968, Z -3.0000, A 0.000, B 0.000, C 0.000 }
gfCNCPoint2[13531] = {X 577.3813, Y 46.6655, Z -3.0000, A 0.000, B 0.000, C 0.000 }
gfCNCPoint2[13532] = {X 572.0983, Y 33.7470, Z -3.0000, A 0.000, B 0.000, C 0.000 }
gfCNCPoint2[13533] = {X 572.0986, Y 40.7327, Z -3.0000, A 0.000, B 0.000, C 0.000 }
gfCNCPoint2[13534] = {X 572.7433, Y 41.4218, Z -3.0000, A 0.000, B 0.000, C 0.000 }
gfCNCPoint2[13535] = {X 573.2263, Y 42.2326, Z -3.0000, A 0.000, B 0.000, C 0.000 }
gfCNCPoint2[13536] = {X 573.5252, Y 43.1277, Z -3.0000, A 0.000, B 0.000, C 0.000 }
gfCNCPoint2[13537] = {X 573.6264, Y 44.0660, Z -3.0000, A 0.000, B 0.000, C 0.000 }
gfCNCPoint2[13538] = {X 573.6264, Y 45.0000, Z -3.0000, A 0.000, B 0.000, C 0.000 }
gfCNCPoint2[13539] = {X 573.5140, Y 45.9884, Z -3.0000, A 0.000, B 0.000, C 0.000 }
gfCNCPoint2[13540] = {X 573.1824, Y 46.9263, Z -3.0000, A 0.000, B 0.000, C 0.000 }
gfCNCPoint2[13541] = {X 572.8094, Y 47.5539, Z -3.0000, A 0.000, B 0.000, C 0.000 }
gfCNCPoint2[13542] = {X 572.3377, Y 48.1113, Z -3.0000, A 0.000, B 0.000, C 0.000 }
gfCNCPoint2[13543] = {X 571.6709, Y 48.6585, Z -3.0000, A 0.000, B 0.000, C 0.000 }
gfCNCPoint2[13544] = {X 570.9102, Y 49.0651, Z -3.0000, A 0.000, B 0.000, C 0.000 }
gfCNCPoint2[13545] = {X 570.0848, Y 49.3155, Z -3.0000, A 0.000, B 0.000, C 0.000 }
gfCNCPoint2[13546] = {X 569.2264, Y 49.4000, Z -3.0000, A 0.000, B 0.000, C 0.000 }
gfCNCPoint2[13547] = {X 562.4443, Y 49.4000, Z -3.0000, A 0.000, B 0.000, C 0.000 }
gfCNCPoint2[13548] = {X 561.4652, Y 49.2897, Z -3.0000, A 0.000, B 0.000, C 0.000 }
gfCNCPoint2[13549] = {X 560.5352, Y 48.9643, Z -3.0000, A 0.000, B 0.000, C 0.000 }
gfCNCPoint2[13550] = {X 559.7009, Y 48.4401, Z -3.0000, A 0.000, B 0.000, C 0.000 }
gfCNCPoint2[13551] = {X 559.0042, Y 47.7434, Z -3.0000, A 0.000, B 0.000, C 0.000 }
gfCNCPoint2[13552] = {X 558.4800, Y 46.9091, Z -3.0000, A 0.000, B 0.000, C 0.000 }
gfCNCPoint2[13553] = {X 558.1546, Y 45.9791, Z -3.0000, A 0.000, B 0.000, C 0.000 }
gfCNCPoint2[13554] = {X 558.0443, Y 45.0000, Z -3.0000, A 0.000, B 0.000, C 0.000 }
gfCNCPoint2[13555] = {X 558.0443, Y 44.0642, Z -3.0000, A 0.000, B 0.000, C 0.000 }
gfCNCPoint2[13556] = {X 558.1487, Y 43.1276, Z -3.0000, A 0.000, B 0.000, C 0.000 }
gfCNCPoint2[13557] = {X 558.4486, Y 42.2342, Z -3.0000, A 0.000, B 0.000, C 0.000 }
gfCNCPoint2[13558] = {X 558.9304, Y 41.4243, Z -3.0000, A 0.000, B 0.000, C 0.000 }
gfCNCPoint2[13559] = {X 559.5724, Y 40.7345, Z -3.0000, A 0.000, B 0.000, C 0.000 }
gfCNCPoint2[13560] = {X 559.5724, Y 9.2675, Z -3.0000, A 0.000, B 0.000, C 0.000 }
gfCNCPoint2[13561] = {X 558.9275, Y 8.5784, Z -3.0000, A 0.000, B 0.000, C 0.000 }
gfCNCPoint2[13562] = {X 558.4445, Y 7.7675, Z -3.0000, A 0.000, B 0.000, C 0.000 }
gfCNCPoint2[13563] = {X 558.1455, Y 6.8723, Z -3.0000, A 0.000, B 0.000, C 0.000 }
gfCNCPoint2[13564] = {X 558.0443, Y 5.9339, Z -3.0000, A 0.000, B 0.000, C 0.000 }
gfCNCPoint2[13565] = {X 558.0443, Y 5.0000, Z -3.0000, A 0.000, B 0.000, C 0.000 }
gfCNCPoint2[13566] = {X 558.1353, Y 4.1097, Z -3.0000, A 0.000, B 0.000, C 0.000 }
gfCNCPoint2[13567] = {X 558.4046, Y 3.2562, Z -3.0000, A 0.000, B 0.000, C 0.000 }
gfCNCPoint2[13568] = {X 558.9155, Y 2.3718, Z -3.0000, A 0.000, B 0.000, C 0.000 }
gfCNCPoint2[13569] = {X 559.6166, Y 1.6290, Z -3.0000, A 0.000, B 0.000, C 0.000 }
gfCNCPoint2[13570] = {X 560.4700, Y 1.0678, Z -3.0000, A 0.000, B 0.000, C 0.000 }
gfCNCPoint2[13571] = {X 561.4298, Y 0.7186, Z -3.0000, A 0.000, B 0.000, C 0.000 }
gfCNCPoint2[13572] = {X 562.4443, Y 0.6000, Z -3.0000, A 0.000, B 0.000, C 0.000 }
gfCNCPoint2[13573] = {X 570.9376, Y 0.6000, Z -3.0000, A 0.000, B 0.000, C 0.000 }
gfCNCPoint2[13574] = {X 571.9520, Y 0.7186, Z -3.0000, A 0.000, B 0.000, C 0.000 }
gfCNCPoint2[13575] = {X 572.9119, Y 1.0678, Z -3.0000, A 0.000, B 0.000, C 0.000 }
gfCNCPoint2[13576] = {X 573.7653, Y 1.6290, Z -3.0000, A 0.000, B 0.000, C 0.000 }
gfCNCPoint2[13577] = {X 574.4664, Y 2.3718, Z -3.0000, A 0.000, B 0.000, C 0.000 }
gfCNCPoint2[13578] = {X 574.9773, Y 3.2562, Z -3.0000, A 0.000, B 0.000, C 0.000 }
gfCNCPoint2[13579] = {X 575.2465, Y 4.1097, Z -3.0000, A 0.000, B 0.000, C 0.000 }
gfCNCPoint2[13580] = {X 575.3376, Y 5.0000, Z -3.0000, A 0.000, B 0.000, C 0.000 }
gfCNCPoint2[13581] = {X 575.3372, Y 5.9910, Z -3.0000, A 0.000, B 0.000, C 0.000 }
gfCNCPoint2[13582] = {X 575.2576, Y 6.7690, Z -3.0000, A 0.000, B 0.000, C 0.000 }
gfCNCPoint2[13583] = {X 575.0416, Y 7.5206, Z -3.0000, A 0.000, B 0.000, C 0.000 }
gfCNCPoint2[13584] = {X 574.6959, Y 8.2221, Z -3.0000, A 0.000, B 0.000, C 0.000 }
gfCNCPoint2[13585] = {X 575.0160, Y 9.0023, Z -3.0000, A 0.000, B 0.000, C 0.000 }
gfCNCPoint2[13586] = {X 581.1911, Y 24.1587, Z -3.0000, A 0.000, B 0.000, C 0.000 }
gfCNCPoint2[13587] = {X 587.7571, Y 8.1002, Z -3.0000, A 0.000, B 0.000, C 0.000 }
gfCNCPoint2[13588] = {X 587.4435, Y 7.4145, Z -3.0000, A 0.000, B 0.000, C 0.000 }
gfCNCPoint2[13589] = {X 587.2515, Y 6.6852, Z -3.0000, A 0.000, B 0.000, C 0.000 }
gfCNCPoint2[13590] = {X 587.1870, Y 5.9339, Z -3.0000, A 0.000, B 0.000, C 0.000 }
gfCNCPoint2[13591] = {X 587.1870, Y 5.0000, Z -3.0000, A 0.000, B 0.000, C 0.000 }
gfCNCPoint2[13592] = {X 587.2780, Y 4.1097, Z -3.0000, A 0.000, B 0.000, C 0.000 }
gfCNCPoint2[13593] = {X 587.5473, Y 3.2562, Z -3.0000, A 0.000, B 0.000, C 0.000 }
gfCNCPoint2[13594] = {X 588.0582, Y 2.3718, Z -3.0000, A 0.000, B 0.000, C 0.000 }
gfCNCPoint2[13595] = {X 588.7592, Y 1.6290, Z -3.0000, A 0.000, B 0.000, C 0.000 }
gfCNCPoint2[13596] = {X 589.6126, Y 1.0678, Z -3.0000, A 0.000, B 0.000, C 0.000 }
gfCNCPoint2[13597] = {X 590.5725, Y 0.7186, Z -3.0000, A 0.000, B 0.000, C 0.000 }
gfCNCPoint2[13598] = {X 591.5870, Y 0.6000, Z -3.0000, A 0.000, B 0.000, C 0.000 }
gfCNCPoint2[13599] = {X 600.0000, Y 0.6000, Z -3.0000, A 0.000, B 0.000, C 0.000 }
gfCNCPoint2[13600] = {X 600.8720, Y 0.6873, Z -3.0000, A 0.000, B 0.000, C 0.000 }
gfCNCPoint2[13601] = {X 601.7094, Y 0.9456, Z -3.0000, A 0.000, B 0.000, C 0.000 }
gfCNCPoint2[13602] = {X 602.4790, Y 1.3648, Z -3.0000, A 0.000, B 0.000, C 0.000 }
gfCNCPoint2[13603] = {X 603.1502, Y 1.9282, Z -3.0000, A 0.000, B 0.000, C 0.000 }
gfCNCPoint2[13604] = {X 603.6965, Y 2.6134, Z -3.0000, A 0.000, B 0.000, C 0.000 }
gfCNCPoint2[13605] = {X 603.6965, Y 1.8141, Z -3.0000, A 0.000, B 0.000, C 0.000 }
gfCNCPoint2[13606] = {X 602.9512, Y 1.1135, Z -3.0000, A 0.000, B 0.000, C 0.000 }
gfCNCPoint2[13607] = {X 602.0762, Y 0.5837, Z -3.0000, A 0.000, B 0.000, C 0.000 }
gfCNCPoint2[13608] = {X 601.1100, Y 0.2479, Z -3.0000, A 0.000, B 0.000, C 0.000 }
gfCNCPoint2[13609] = {X 600.0951, Y 0.1209, Z -3.0000, A 0.000, B 0.000, C 0.000 }
gfCNCPoint2[13610] = {X 600.0948, Y -0.0187, Z -3.0000, A 0.000, B 0.000, C 0.000 }
gfCNCPoint2[13611] = {X 600.0672, Y -0.0698, Z -3.0000, A 0.000, B 0.000, C 0.000 }
gfCNCPoint2[13612] = {X 600.0148, Y -0.0950, Z -3.0000, A 0.000, B 0.000, C 0.000 }
gfCNCPoint2[13613] = {X 580.1328, Y -0.0950, Z -3.0000, A 0.000, B 0.000, C 0.000 }
gfCNCPoint2[13614] = {X 580.1328, Y 4.7050, Z -3.0000, A 0.000, B 0.000, C 0.000 }
gfCNCPoint2[13615] = {X 580.1364, Y 4.8525, Z -3.0000, A 0.000, B 0.000, C 0.000 }
gfCNCPoint2[13616] = {X 580.1376, Y 5.0000, Z -3.0000, A 0.000, B 0.000, C 0.000 }
gfCNCPoint2[13617] = {X 580.1368, Y 6.0531, Z -3.0000, A 0.000, B 0.000, C 0.000 }
gfCNCPoint2[13618] = {X 580.0607, Y 7.1209, Z -3.0000, A 0.000, B 0.000, C 0.000 }
gfCNCPoint2[13619] = {X 579.8611, Y 8.1726, Z -3.0000, A 0.000, B 0.000, C 0.000 }
gfCNCPoint2[13620] = {X 581.1990, Y 11.4566, Z -3.0000, A 0.000, B 0.000, C 0.000 }
gfCNCPoint2[13621] = {X 582.6185, Y 7.9850, Z -3.0000, A 0.000, B 0.000, C 0.000 }
gfCNCPoint2[13622] = {X 582.4489, Y 6.9997, Z -3.0000, A 0.000, B 0.000, C 0.000 }
gfCNCPoint2[13623] = {X 582.3872, Y 6.0018, Z -3.0000, A 0.000, B 0.000, C 0.000 }
gfCNCPoint2[13624] = {X 582.3870, Y 5.0000, Z -3.0000, A 0.000, B 0.000, C 0.000 }
gfCNCPoint2[13625] = {X 582.3881, Y 4.8525, Z -3.0000, A 0.000, B 0.000, C 0.000 }
gfCNCPoint2[13626] = {X 582.3917, Y 4.7050, Z -3.0000, A 0.000, B 0.000, C 0.000 }
gfCNCPoint2[13627] = {X 580.1328, Y 4.7050, Z -3.0000, A 0.000, B 0.000, C 0.000 }
gfCNCPoint2[13628] = {X 580.1328, Y 2.3050, Z -3.0000, A 0.000, B 0.000, C 0.000 }
gfCNCPoint2[13629] = {X 577.1807, Y 2.3050, Z -3.0000, A 0.000, B 0.000, C 0.000 }
gfCNCPoint2[13630] = {X 577.5740, Y 3.5175, Z -3.0000, A 0.000, B 0.000, C 0.000 }
gfCNCPoint2[13631] = {X 577.7341, Y 4.7820, Z -3.0000, A 0.000, B 0.000, C 0.000 }
gfCNCPoint2[13632] = {X 577.7367, Y 4.8910, Z -3.0000, A 0.000, B 0.000, C 0.000 }
gfCNCPoint2[13633] = {X 577.7376, Y 5.0000, Z -3.0000, A 0.000, B 0.000, C 0.000 }
gfCNCPoint2[13634] = {X 577.7370, Y 6.0220, Z -3.0000, A 0.000, B 0.000, C 0.000 }
gfCNCPoint2[13635] = {X 577.6237, Y 7.1733, Z -3.0000, A 0.000, B 0.000, C 0.000 }
gfCNCPoint2[13636] = {X 577.3168, Y 8.2888, Z -3.0000, A 0.000, B 0.000, C 0.000 }
gfCNCPoint2[13637] = {X 581.1951, Y 17.8077, Z -3.0000, A 0.000, B 0.000, C 0.000 }
gfCNCPoint2[13638] = {X 585.1516, Y 8.1310, Z -3.0000, A 0.000, B 0.000, C 0.000 }
gfCNCPoint2[13639] = {X 584.8835, Y 7.0759, Z -3.0000, A 0.000, B 0.000, C 0.000 }
gfCNCPoint2[13640] = {X 584.7872, Y 5.9914, Z -3.0000, A 0.000, B 0.000, C 0.000 }
gfCNCPoint2[13641] = {X 584.7870, Y 5.0000, Z -3.0000, A 0.000, B 0.000, C 0.000 }
gfCNCPoint2[13642] = {X 584.7878, Y 4.8910, Z -3.0000, A 0.000, B 0.000, C 0.000 }
gfCNCPoint2[13643] = {X 584.7904, Y 4.7820, Z -3.0000, A 0.000, B 0.000, C 0.000 }
gfCNCPoint2[13644] = {X 584.9505, Y 3.5175, Z -3.0000, A 0.000, B 0.000, C 0.000 }
gfCNCPoint2[13645] = {X 585.3438, Y 2.3050, Z -3.0000, A 0.000, B 0.000, C 0.000 }
gfCNCPoint2[13646] = {X 580.1328, Y 2.3050, Z -3.0000, A 0.000, B 0.000, C 0.000 }
gfCNCPoint2[13647] = {X 580.1328, Y -0.0950, Z -3.0000, A 0.000, B 0.000, C 0.000 }
gfCNCPoint2[13648] = {X 351.5638, Y -0.0950, Z -3.0000, A 0.000, B 0.000, C 0.000 }
gfCNCPoint2[13649] = {X 351.4053, Y -0.1244, Z -3.0000, A 0.000, B 0.000, C 0.000 }
gfCNCPoint2[13650] = {X 348.9098, Y -0.4707, Z -3.0000, A 0.000, B 0.000, C 0.000 }
gfCNCPoint2[13651] = {X 346.3929, Y -0.5816, Z -3.0000, A 0.000, B 0.000, C 0.000 }
gfCNCPoint2[13652] = {X 343.8766, Y -0.4560, Z -3.0000, A 0.000, B 0.000, C 0.000 }
gfCNCPoint2[13653] = {X 341.3832, Y -0.0950, Z -3.0000, A 0.000, B 0.000, C 0.000 }
gfCNCPoint2[13654] = {X -0.0148, Y -0.0950, Z -3.0000, A 0.000, B 0.000, C 0.000 }
gfCNCPoint2[13655] = {X -0.0672, Y -0.0698, Z -3.0000, A 0.000, B 0.000, C 0.000 }
gfCNCPoint2[13656] = {X -0.0948, Y -0.0187, Z -3.0000, A 0.000, B 0.000, C 0.000 }
gfCNCPoint2[13657] = {X -0.0965, Y 0.8569, Z -3.0000, A 0.000, B 0.000, C 0.000 }
gfCNCPoint2[13658] = {X -0.0965, Y 8.7891, Z -3.0000, A 0.000, B 0.000, C 0.000 }
gfCNCPoint2[13659] = {X -0.7633, Y 8.9979, Z -3.0000, A 0.000, B 0.000, C 0.000 }
gfCNCPoint2[13660] = {X -1.3934, Y 9.2998, Z -3.0000, A 0.000, B 0.000, C 0.000 }
gfCNCPoint2[13661] = {X -1.9904, Y 9.6404, Z -3.0000, A 0.000, B 0.000, C 0.000 }
gfCNCPoint2[13662] = {X -2.6455, Y 10.0884, Z -3.0000, A 0.000, B 0.000, C 0.000 }
gfCNCPoint2[13663] = {X -3.2192, Y 10.6366, Z -3.0000, A 0.000, B 0.000, C 0.000 }
gfCNCPoint2[13664] = {X -3.6965, Y 11.2706, Z -3.0000, A 0.000, B 0.000, C 0.000 }
gfCNCPoint2[13665] = {X -3.6965, Y 12.3461, Z -3.0000, A 0.000, B 0.000, C 0.000 }
gfCNCPoint2[13666] = {X -3.2332, Y 11.4383, Z -3.0000, A 0.000, B 0.000, C 0.000 }
gfCNCPoint2[13667] = {X -2.5734, Y 10.6615, Z -3.0000, A 0.000, B 0.000, C 0.000 }
gfCNCPoint2[13668] = {X -1.7526, Y 10.0573, Z -3.0000, A 0.000, B 0.000, C 0.000 }
gfCNCPoint2[13669] = {X -1.0994, Y 9.6852, Z -3.0000, A 0.000, B 0.000, C 0.000 }
gfCNCPoint2[13670] = {X -0.1608, Y 9.3012, Z -3.0000, A 0.000, B 0.000, C 0.000 }
gfCNCPoint2[13671] = {X 0.8408, Y 9.1423, Z -3.0000, A 0.000, B 0.000, C 0.000 }
gfCNCPoint2[13672] = {X 1.8522, Y 9.2169, Z -3.0000, A 0.000, B 0.000, C 0.000 }
gfCNCPoint2[13673] = {X 2.2366, Y 9.3086, Z -3.0000, A 0.000, B 0.000, C 0.000 }
gfCNCPoint2[13674] = {X 2.6112, Y 9.4344, Z -3.0000, A 0.000, B 0.000, C 0.000 }
gfCNCPoint2[13675] = {X 3.3793, Y 9.0771, Z -3.0000, A 0.000, B 0.000, C 0.000 }
gfCNCPoint2[13676] = {X 4.1685, Y 8.7694, Z -3.0000, A 0.000, B 0.000, C 0.000 }
gfCNCPoint2[13677] = {X 6.0858, Y 8.0984, Z -3.0000, A 0.000, B 0.000, C 0.000 }
gfCNCPoint2[13678] = {X 8.0538, Y 7.5953, Z -3.0000, A 0.000, B 0.000, C 0.000 }
gfCNCPoint2[13679] = {X 10.0579, Y 7.2638, Z -3.0000, A 0.000, B 0.000, C 0.000 }
gfCNCPoint2[13680] = {X 12.0831, Y 7.1063, Z -3.0000, A 0.000, B 0.000, C 0.000 }
gfCNCPoint2[13681] = {X 14.1143, Y 7.1241, Z -3.0000, A 0.000, B 0.000, C 0.000 }
gfCNCPoint2[13682] = {X 16.1365, Y 7.3170, Z -3.0000, A 0.000, B 0.000, C 0.000 }
gfCNCPoint2[13683] = {X 16.5415, Y 7.3732, Z -3.0000, A 0.000, B 0.000, C 0.000 }
gfCNCPoint2[13684] = {X 18.2855, Y 7.7306, Z -3.0000, A 0.000, B 0.000, C 0.000 }
gfCNCPoint2[13685] = {X 19.9843, Y 8.2631, Z -3.0000, A 0.000, B 0.000, C 0.000 }
gfCNCPoint2[13686] = {X 21.6203, Y 8.9650, Z -3.0000, A 0.000, B 0.000, C 0.000 }
gfCNCPoint2[13687] = {X 23.1768, Y 9.8292, Z -3.0000, A 0.000, B 0.000, C 0.000 }
gfCNCPoint2[13688] = {X 24.6376, Y 10.8467, Z -3.0000, A 0.000, B 0.000, C 0.000 }
gfCNCPoint2[13689] = {X 25.7299, Y 11.8020, Z -3.0000, A 0.000, B 0.000, C 0.000 }
gfCNCPoint2[13690] = {X 26.7097, Y 12.8724, Z -3.0000, A 0.000, B 0.000, C 0.000 }
gfCNCPoint2[13691] = {X 27.5647, Y 14.0448, Z -3.0000, A 0.000, B 0.000, C 0.000 }
gfCNCPoint2[13692] = {X 28.2846, Y 15.3048, Z -3.0000, A 0.000, B 0.000, C 0.000 }
gfCNCPoint2[13693] = {X 28.8604, Y 16.6368, Z -3.0000, A 0.000, B 0.000, C 0.000 }
gfCNCPoint2[13694] = {X 29.3370, Y 18.3013, Z -3.0000, A 0.000, B 0.000, C 0.000 }
gfCNCPoint2[13695] = {X 29.6197, Y 20.0094, Z -3.0000, A 0.000, B 0.000, C 0.000 }
gfCNCPoint2[13696] = {X 29.7049, Y 21.7387, Z -3.0000, A 0.000, B 0.000, C 0.000 }
gfCNCPoint2[13697] = {X 29.5914, Y 23.4664, Z -3.0000, A 0.000, B 0.000, C 0.000 }
gfCNCPoint2[13698] = {X 29.2808, Y 25.1696, Z -3.0000, A 0.000, B 0.000, C 0.000 }
gfCNCPoint2[13699] = {X 28.7896, Y 26.7454, Z -3.0000, A 0.000, B 0.000, C 0.000 }
gfCNCPoint2[13700] = {X 28.0828, Y 28.2369, Z -3.0000, A 0.000, B 0.000, C 0.000 }
gfCNCPoint2[13701] = {X 27.1743, Y 29.6149, Z -3.0000, A 0.000, B 0.000, C 0.000 }
gfCNCPoint2[13702] = {X 26.3573, Y 30.5721, Z -3.0000, A 0.000, B 0.000, C 0.000 }
gfCNCPoint2[13703] = {X 25.4427, Y 31.4365, Z -3.0000, A 0.000, B 0.000, C 0.000 }
gfCNCPoint2[13704] = {X 25.6933, Y 31.5321, Z -3.0000, A 0.000, B 0.000, C 0.000 }
gfCNCPoint2[13705] = {X 25.9376, Y 31.6428, Z -3.0000, A 0.000, B 0.000, C 0.000 }
gfCNCPoint2[13706] = {X 26.3180, Y 31.8533, Z -3.0000, A 0.000, B 0.000, C 0.000 }
gfCNCPoint2[13707] = {X 26.6757, Y 32.1002, Z -3.0000, A 0.000, B 0.000, C 0.000 }
gfCNCPoint2[13708] = {X 26.9951, Y 32.3698, Z -3.0000, A 0.000, B 0.000, C 0.000 }
gfCNCPoint2[13709] = {X 27.2875, Y 32.6685, Z -3.0000, A 0.000, B 0.000, C 0.000 }
gfCNCPoint2[13710] = {X 27.6591, Y 33.1492, Z -3.0000, A 0.000, B 0.000, C 0.000 }
gfCNCPoint2[13711] = {X 27.9609, Y 33.6766, Z -3.0000, A 0.000, B 0.000, C 0.000 }
gfCNCPoint2[13712] = {X 30.9820, Y 39.9182, Z -3.0000, A 0.000, B 0.000, C 0.000 }
gfCNCPoint2[13713] = {X 31.3085, Y 40.8441, Z -3.0000, A 0.000, B 0.000, C 0.000 }
gfCNCPoint2[13714] = {X 31.4215, Y 41.8194, Z -3.0000, A 0.000, B 0.000, C 0.000 }
gfCNCPoint2[13715] = {X 31.3155, Y 42.7955, Z -3.0000, A 0.000, B 0.000, C 0.000 }
gfCNCPoint2[13716] = {X 30.9956, Y 43.7238, Z -3.0000, A 0.000, B 0.000, C 0.000 }
gfCNCPoint2[13717] = {X 30.4779, Y 44.5580, Z -3.0000, A 0.000, B 0.000, C 0.000 }
gfCNCPoint2[13718] = {X 29.7880, Y 45.2567, Z -3.0000, A 0.000, B 0.000, C 0.000 }
gfCNCPoint2[13719] = {X 29.2517, Y 45.6903, Z -3.0000, A 0.000, B 0.000, C 0.000 }
gfCNCPoint2[13720] = {X 28.5403, Y 46.1588, Z -3.0000, A 0.000, B 0.000, C 0.000 }
gfCNCPoint2[13721] = {X 27.7522, Y 46.4820, Z -3.0000, A 0.000, B 0.000, C 0.000 }
gfCNCPoint2[13722] = {X 26.9167, Y 46.6478, Z -3.0000, A 0.000, B 0.000, C 0.000 }
gfCNCPoint2[13723] = {X 26.0650, Y 46.6502, Z -3.0000, A 0.000, B 0.000, C 0.000 }
gfCNCPoint2[13724] = {X 25.2286, Y 46.4891, Z -3.0000, A 0.000, B 0.000, C 0.000 }
gfCNCPoint2[13725] = {X 23.6560, Y 47.3292, Z -3.0000, A 0.000, B 0.000, C 0.000 }
gfCNCPoint2[13726] = {X 22.0332, Y 48.0678, Z -3.0000, A 0.000, B 0.000, C 0.000 }
gfCNCPoint2[13727] = {X 20.3668, Y 48.7018, Z -3.0000, A 0.000, B 0.000, C 0.000 }
gfCNCPoint2[13728] = {X 19.6694, Y 48.9423, Z -3.0000, A 0.000, B 0.000, C 0.000 }
gfCNCPoint2[13729] = {X 17.4685, Y 49.5493, Z -3.0000, A 0.000, B 0.000, C 0.000 }
gfCNCPoint2[13730] = {X 15.2180, Y 49.9342, Z -3.0000, A 0.000, B 0.000, C 0.000 }
gfCNCPoint2[13731] = {X 12.9404, Y 50.0930, Z -3.0000, A 0.000, B 0.000, C 0.000 }
gfCNCPoint2[13732] = {X 10.6582, Y 50.0242, Z -3.0000, A 0.000, B 0.000, C 0.000 }
gfCNCPoint2[13733] = {X 8.3943, Y 49.7285, Z -3.0000, A 0.000, B 0.000, C 0.000 }
gfCNCPoint2[13734] = {X 6.6780, Y 49.3394, Z -3.0000, A 0.000, B 0.000, C 0.000 }
gfCNCPoint2[13735] = {X 5.0103, Y 48.7771, Z -3.0000, A 0.000, B 0.000, C 0.000 }
gfCNCPoint2[13736] = {X 3.4087, Y 48.0476, Z -3.0000, A 0.000, B 0.000, C 0.000 }
gfCNCPoint2[13737] = {X 2.3351, Y 47.4409, Z -3.0000, A 0.000, B 0.000, C 0.000 }
gfCNCPoint2[13738] = {X 1.3077, Y 46.7589, Z -3.0000, A 0.000, B 0.000, C 0.000 }
gfCNCPoint2[13739] = {X -0.0252, Y 45.6857, Z -3.0000, A 0.000, B 0.000, C 0.000 }
gfCNCPoint2[13740] = {X -1.2102, Y 44.4510, Z -3.0000, A 0.000, B 0.000, C 0.000 }
gfCNCPoint2[13741] = {X -2.2276, Y 43.0750, Z -3.0000, A 0.000, B 0.000, C 0.000 }
gfCNCPoint2[13742] = {X -3.0610, Y 41.5804, Z -3.0000, A 0.000, B 0.000, C 0.000 }
gfCNCPoint2[13743] = {X -3.6965, Y 39.9915, Z -3.0000, A 0.000, B 0.000, C 0.000 }
gfCNCPoint2[13744] = {X -3.6965, Y 41.3423, Z -3.0000, A 0.000, B 0.000, C 0.000 }
gfCNCPoint2[13745] = {X -3.0077, Y 42.7159, Z -3.0000, A 0.000, B 0.000, C 0.000 }
gfCNCPoint2[13746] = {X -2.1710, Y 44.0048, Z -3.0000, A 0.000, B 0.000, C 0.000 }
gfCNCPoint2[13747] = {X -1.1966, Y 45.1930, Z -3.0000, A 0.000, B 0.000, C 0.000 }
gfCNCPoint2[13748] = {X -0.0965, Y 46.2659, Z -3.0000, A 0.000, B 0.000, C 0.000 }
gfCNCPoint2[13749] = {X -0.0965, Y 99.1431, Z -3.0000, A 0.000, B 0.000, C 0.000 }
gfCNCPoint2[13750] = {X -0.0948, Y 100.0187, Z -3.0000, A 0.000, B 0.000, C 0.000 }
gfCNCPoint2[13751] = {X -0.0672, Y 100.0698, Z -3.0000, A 0.000, B 0.000, C 0.000 }
gfCNCPoint2[13752] = {X -0.0148, Y 100.0950, Z -3.0000, A 0.000, B 0.000, C 0.000 }
gfCNCPoint2[13753] = {X 120.5926, Y 100.0950, Z -3.0000, A 0.000, B 0.000, C 0.000 }
gfCNCPoint2[13754] = {X 121.0613, Y 100.8812, Z -3.0000, A 0.000, B 0.000, C 0.000 }
gfCNCPoint2[13755] = {X 121.6686, Y 101.5660, Z -3.0000, A 0.000, B 0.000, C 0.000 }
gfCNCPoint2[13756] = {X 122.3932, Y 102.1254, Z -3.0000, A 0.000, B 0.000, C 0.000 }
gfCNCPoint2[13757] = {X 123.2094, Y 102.5396, Z -3.0000, A 0.000, B 0.000, C 0.000 }
gfCNCPoint2[13758] = {X 124.0887, Y 102.7942, Z -3.0000, A 0.000, B 0.000, C 0.000 }
gfCNCPoint2[13759] = {X 125.0000, Y 102.8800, Z -3.0000, A 0.000, B 0.000, C 0.000 }
gfCNCPoint2[13760] = {X 143.7791, Y 102.8800, Z -3.0000, A 0.000, B 0.000, C 0.000 }
gfCNCPoint2[13761] = {X 144.6904, Y 102.7942, Z -3.0000, A 0.000, B 0.000, C 0.000 }
gfCNCPoint2[13762] = {X 145.5697, Y 102.5396, Z -3.0000, A 0.000, B 0.000, C 0.000 }
gfCNCPoint2[13763] = {X 146.3859, Y 102.1254, Z -3.0000, A 0.000, B 0.000, C 0.000 }
gfCNCPoint2[13764] = {X 147.1105, Y 101.5660, Z -3.0000, A 0.000, B 0.000, C 0.000 }
gfCNCPoint2[13765] = {X 147.7178, Y 100.8812, Z -3.0000, A 0.000, B 0.000, C 0.000 }
gfCNCPoint2[13766] = {X 148.1866, Y 100.0950, Z -3.0000, A 0.000, B 0.000, C 0.000 }
gfCNCPoint2[13767] = {X 150.8373, Y 100.0950, Z -3.0000, A 0.000, B 0.000, C 0.000 }
gfCNCPoint2[13768] = {X 150.8373, Y 95.2950, Z -3.0000, A 0.000, B 0.000, C 0.000 }
gfCNCPoint2[13769] = {X 187.9257, Y 95.2950, Z -3.0000, A 0.000, B 0.000, C 0.000 }
gfCNCPoint2[13770] = {X 187.9777, Y 95.0990, Z -3.0000, A 0.000, B 0.000, C 0.000 }
gfCNCPoint2[13771] = {X 188.0352, Y 94.9045, Z -3.0000, A 0.000, B 0.000, C 0.000 }
gfCNCPoint2[13772] = {X 187.2619, Y 94.0602, Z -3.0000, A 0.000, B 0.000, C 0.000 }
gfCNCPoint2[13773] = {X 151.4055, Y 94.0602, Z -3.0000, A 0.000, B 0.000, C 0.000 }
gfCNCPoint2[13774] = {X 150.7055, Y 94.8358, Z -3.0000, A 0.000, B 0.000, C 0.000 }
gfCNCPoint2[13775] = {X 150.7752, Y 95.0643, Z -3.0000, A 0.000, B 0.000, C 0.000 }
gfCNCPoint2[13776] = {X 150.8373, Y 95.2950, Z -3.0000, A 0.000, B 0.000, C 0.000 }
gfCNCPoint2[13777] = {X 150.8373, Y 97.6950, Z -3.0000, A 0.000, B 0.000, C 0.000 }
gfCNCPoint2[13778] = {X 190.1070, Y 97.6950, Z -3.0000, A 0.000, B 0.000, C 0.000 }
gfCNCPoint2[13779] = {X 190.1070, Y 97.0659, Z -3.0000, A 0.000, B 0.000, C 0.000 }
gfCNCPoint2[13780] = {X 190.1938, Y 96.1495, Z -3.0000, A 0.000, B 0.000, C 0.000 }
gfCNCPoint2[13781] = {X 190.4511, Y 95.2657, Z -3.0000, A 0.000, B 0.000, C 0.000 }
gfCNCPoint2[13782] = {X 190.8699, Y 94.4460, Z -3.0000, A 0.000, B 0.000, C 0.000 }
gfCNCPoint2[13783] = {X 188.3182, Y 91.6602, Z -3.0000, A 0.000, B 0.000, C 0.000 }
gfCNCPoint2[13784] = {X 150.3387, Y 91.6602, Z -3.0000, A 0.000, B 0.000, C 0.000 }
gfCNCPoint2[13785] = {X 147.8635, Y 94.4025, Z -3.0000, A 0.000, B 0.000, C 0.000 }
gfCNCPoint2[13786] = {X 148.2976, Y 95.2328, Z -3.0000, A 0.000, B 0.000, C 0.000 }
gfCNCPoint2[13787] = {X 148.5661, Y 96.1304, Z -3.0000, A 0.000, B 0.000, C 0.000 }
gfCNCPoint2[13788] = {X 148.6591, Y 97.0627, Z -3.0000, A 0.000, B 0.000, C 0.000 }
gfCNCPoint2[13789] = {X 148.6591, Y 97.6950, Z -3.0000, A 0.000, B 0.000, C 0.000 }
gfCNCPoint2[13790] = {X 150.8373, Y 97.6950, Z -3.0000, A 0.000, B 0.000, C 0.000 }
gfCNCPoint2[13791] = {X 150.8373, Y 100.0950, Z -3.0000, A 0.000, B 0.000, C 0.000 }
gfCNCPoint2[13792] = {X 190.5795, Y 100.0950, Z -3.0000, A 0.000, B 0.000, C 0.000 }
gfCNCPoint2[13793] = {X 191.0483, Y 100.8812, Z -3.0000, A 0.000, B 0.000, C 0.000 }
gfCNCPoint2[13794] = {X 191.6556, Y 101.5660, Z -3.0000, A 0.000, B 0.000, C 0.000 }
gfCNCPoint2[13795] = {X 192.3801, Y 102.1254, Z -3.0000, A 0.000, B 0.000, C 0.000 }
gfCNCPoint2[13796] = {X 193.1964, Y 102.5396, Z -3.0000, A 0.000, B 0.000, C 0.000 }
gfCNCPoint2[13797] = {X 194.0756, Y 102.7942, Z -3.0000, A 0.000, B 0.000, C 0.000 }
gfCNCPoint2[13798] = {X 194.9870, Y 102.8800, Z -3.0000, A 0.000, B 0.000, C 0.000 }
gfCNCPoint2[13799] = {X 212.6141, Y 102.8800, Z -3.0000, A 0.000, B 0.000, C 0.000 }
gfCNCPoint2[13800] = {X 213.0066, Y 102.8642, Z -3.0000, A 0.000, B 0.000, C 0.000 }
gfCNCPoint2[13801] = {X 213.3966, Y 102.8169, Z -3.0000, A 0.000, B 0.000, C 0.000 }
gfCNCPoint2[13802] = {X 213.7865, Y 102.8642, Z -3.0000, A 0.000, B 0.000, C 0.000 }
gfCNCPoint2[13803] = {X 214.1790, Y 102.8800, Z -3.0000, A 0.000, B 0.000, C 0.000 }
gfCNCPoint2[13804] = {X 233.4798, Y 102.8800, Z -3.0000, A 0.000, B 0.000, C 0.000 }
gfCNCPoint2[13805] = {X 234.3911, Y 102.7942, Z -3.0000, A 0.000, B 0.000, C 0.000 }
gfCNCPoint2[13806] = {X 235.2704, Y 102.5396, Z -3.0000, A 0.000, B 0.000, C 0.000 }
gfCNCPoint2[13807] = {X 236.0866, Y 102.1254, Z -3.0000, A 0.000, B 0.000, C 0.000 }
gfCNCPoint2[13808] = {X 236.8111, Y 101.5660, Z -3.0000, A 0.000, B 0.000, C 0.000 }
gfCNCPoint2[13809] = {X 237.4185, Y 100.8812, Z -3.0000, A 0.000, B 0.000, C 0.000 }
gfCNCPoint2[13810] = {X 237.8872, Y 100.0950, Z -3.0000, A 0.000, B 0.000, C 0.000 }
gfCNCPoint2[13811] = {X 261.4771, Y 100.0950, Z -3.0000, A 0.000, B 0.000, C 0.000 }
gfCNCPoint2[13812] = {X 261.4771, Y 90.4950, Z -3.0000, A 0.000, B 0.000, C 0.000 }
gfCNCPoint2[13813] = {X 266.0962, Y 90.4950, Z -3.0000, A 0.000, B 0.000, C 0.000 }
gfCNCPoint2[13814] = {X 266.1752, Y 90.3747, Z -3.0000, A 0.000, B 0.000, C 0.000 }
gfCNCPoint2[13815] = {X 266.2556, Y 90.2554, Z -3.0000, A 0.000, B 0.000, C 0.000 }
gfCNCPoint2[13816] = {X 263.5091, Y 89.1787, Z -3.0000, A 0.000, B 0.000, C 0.000 }
gfCNCPoint2[13817] = {X 261.4771, Y 90.4950, Z -3.0000, A 0.000, B 0.000, C 0.000 }
gfCNCPoint2[13818] = {X 261.4771, Y 92.8950, Z -3.0000, A 0.000, B 0.000, C 0.000 }
gfCNCPoint2[13819] = {X 267.4974, Y 92.8950, Z -3.0000, A 0.000, B 0.000, C 0.000 }
gfCNCPoint2[13820] = {X 267.8429, Y 92.2375, Z -3.0000, A 0.000, B 0.000, C 0.000 }
gfCNCPoint2[13821] = {X 268.2378, Y 91.6085, Z -3.0000, A 0.000, B 0.000, C 0.000 }
gfCNCPoint2[13822] = {X 269.1700, Y 90.4463, Z -3.0000, A 0.000, B 0.000, C 0.000 }
gfCNCPoint2[13823] = {X 270.2694, Y 89.4409, Z -3.0000, A 0.000, B 0.000, C 0.000 }
gfCNCPoint2[13824] = {X 270.2694, Y 89.2510, Z -3.0000, A 0.000, B 0.000, C 0.000 }
gfCNCPoint2[13825] = {X 263.2382, Y 86.4947, Z -3.0000, A 0.000, B 0.000, C 0.000 }
gfCNCPoint2[13826] = {X 253.3572, Y 92.8950, Z -3.0000, A 0.000, B 0.000, C 0.000 }
gfCNCPoint2[13827] = {X 261.4771, Y 92.8950, Z -3.0000, A 0.000, B 0.000, C 0.000 }
gfCNCPoint2[13828] = {X 261.4771, Y 95.2950, Z -3.0000, A 0.000, B 0.000, C 0.000 }
gfCNCPoint2[13829] = {X 269.1714, Y 95.2950, Z -3.0000, A 0.000, B 0.000, C 0.000 }
gfCNCPoint2[13830] = {X 269.5516, Y 94.1744, Z -3.0000, A 0.000, B 0.000, C 0.000 }
gfCNCPoint2[13831] = {X 270.1082, Y 93.1303, Z -3.0000, A 0.000, B 0.000, C 0.000 }
gfCNCPoint2[13832] = {X 270.8267, Y 92.1901, Z -3.0000, A 0.000, B 0.000, C 0.000 }
gfCNCPoint2[13833] = {X 271.6880, Y 91.3787, Z -3.0000, A 0.000, B 0.000, C 0.000 }
gfCNCPoint2[13834] = {X 272.6694, Y 90.7176, Z -3.0000, A 0.000, B 0.000, C 0.000 }
gfCNCPoint2[13835] = {X 272.6694, Y 87.6139, Z -3.0000, A 0.000, B 0.000, C 0.000 }
gfCNCPoint2[13836] = {X 262.9673, Y 83.8107, Z -3.0000, A 0.000, B 0.000, C 0.000 }
gfCNCPoint2[13837] = {X 245.2372, Y 95.2950, Z -3.0000, A 0.000, B 0.000, C 0.000 }
gfCNCPoint2[13838] = {X 261.4771, Y 95.2950, Z -3.0000, A 0.000, B 0.000, C 0.000 }
gfCNCPoint2[13839] = {X 261.4771, Y 97.6950, Z -3.0000, A 0.000, B 0.000, C 0.000 }
gfCNCPoint2[13840] = {X 271.3527, Y 97.6950, Z -3.0000, A 0.000, B 0.000, C 0.000 }
gfCNCPoint2[13841] = {X 271.3529, Y 97.0186, Z -3.0000, A 0.000, B 0.000, C 0.000 }
gfCNCPoint2[13842] = {X 271.4810, Y 95.9545, Z -3.0000, A 0.000, B 0.000, C 0.000 }
gfCNCPoint2[13843] = {X 271.8382, Y 94.9440, Z -3.0000, A 0.000, B 0.000, C 0.000 }
gfCNCPoint2[13844] = {X 272.4073, Y 94.0359, Z -3.0000, A 0.000, B 0.000, C 0.000 }
gfCNCPoint2[13845] = {X 273.1610, Y 93.2739, Z -3.0000, A 0.000, B 0.000, C 0.000 }
gfCNCPoint2[13846] = {X 274.0629, Y 92.6949, Z -3.0000, A 0.000, B 0.000, C 0.000 }
gfCNCPoint2[13847] = {X 275.0694, Y 92.3266, Z -3.0000, A 0.000, B 0.000, C 0.000 }
gfCNCPoint2[13848] = {X 275.0694, Y 85.9769, Z -3.0000, A 0.000, B 0.000, C 0.000 }
gfCNCPoint2[13849] = {X 262.6986, Y 81.1276, Z -3.0000, A 0.000, B 0.000, C 0.000 }
gfCNCPoint2[13850] = {X 262.5777, Y 81.2036, Z -3.0000, A 0.000, B 0.000, C 0.000 }
gfCNCPoint2[13851] = {X 238.3585, Y 96.8910, Z -3.0000, A 0.000, B 0.000, C 0.000 }
gfCNCPoint2[13852] = {X 238.3598, Y 97.0659, Z -3.0000, A 0.000, B 0.000, C 0.000 }
gfCNCPoint2[13853] = {X 238.3598, Y 97.6950, Z -3.0000, A 0.000, B 0.000, C 0.000 }
gfCNCPoint2[13854] = {X 261.4771, Y 97.6950, Z -3.0000, A 0.000, B 0.000, C 0.000 }
gfCNCPoint2[13855] = {X 261.4771, Y 100.0950, Z -3.0000, A 0.000, B 0.000, C 0.000 }
gfCNCPoint2[13856] = {X 271.8252, Y 100.0950, Z -3.0000, A 0.000, B 0.000, C 0.000 }
gfCNCPoint2[13857] = {X 272.2940, Y 100.8812, Z -3.0000, A 0.000, B 0.000, C 0.000 }
gfCNCPoint2[13858] = {X 272.9013, Y 101.5660, Z -3.0000, A 0.000, B 0.000, C 0.000 }
gfCNCPoint2[13859] = {X 273.6259, Y 102.1254, Z -3.0000, A 0.000, B 0.000, C 0.000 }
gfCNCPoint2[13860] = {X 274.4421, Y 102.5396, Z -3.0000, A 0.000, B 0.000, C 0.000 }
gfCNCPoint2[13861] = {X 275.3214, Y 102.7942, Z -3.0000, A 0.000, B 0.000, C 0.000 }
gfCNCPoint2[13862] = {X 276.2327, Y 102.8800, Z -3.0000, A 0.000, B 0.000, C 0.000 }
gfCNCPoint2[13863] = {X 292.7731, Y 102.8800, Z -3.0000, A 0.000, B 0.000, C 0.000 }
gfCNCPoint2[13864] = {X 293.6844, Y 102.7942, Z -3.0000, A 0.000, B 0.000, C 0.000 }
gfCNCPoint2[13865] = {X 294.5637, Y 102.5396, Z -3.0000, A 0.000, B 0.000, C 0.000 }
gfCNCPoint2[13866] = {X 295.3799, Y 102.1254, Z -3.0000, A 0.000, B 0.000, C 0.000 }
gfCNCPoint2[13867] = {X 296.1044, Y 101.5660, Z -3.0000, A 0.000, B 0.000, C 0.000 }
gfCNCPoint2[13868] = {X 296.7118, Y 100.8812, Z -3.0000, A 0.000, B 0.000, C 0.000 }
gfCNCPoint2[13869] = {X 297.1805, Y 100.0950, Z -3.0000, A 0.000, B 0.000, C 0.000 }
gfCNCPoint2[13870] = {X 319.1363, Y 100.0950, Z -3.0000, A 0.000, B 0.000, C 0.000 }
gfCNCPoint2[13871] = {X 321.4384, Y 100.8673, Z -3.0000, A 0.000, B 0.000, C 0.000 }
gfCNCPoint2[13872] = {X 323.7829, Y 101.4990, Z -3.0000, A 0.000, B 0.000, C 0.000 }
gfCNCPoint2[13873] = {X 326.1614, Y 101.9878, Z -3.0000, A 0.000, B 0.000, C 0.000 }
gfCNCPoint2[13874] = {X 329.6397, Y 102.5402, Z -3.0000, A 0.000, B 0.000, C 0.000 }
gfCNCPoint2[13875] = {X 333.1371, Y 102.9556, Z -3.0000, A 0.000, B 0.000, C 0.000 }
gfCNCPoint2[13876] = {X 336.6481, Y 103.2334, Z -3.0000, A 0.000, B 0.000, C 0.000 }
gfCNCPoint2[13877] = {X 342.8091, Y 103.5154, Z -3.0000, A 0.000, B 0.000, C 0.000 }
gfCNCPoint2[13878] = {X 348.9760, Y 103.5920, Z -3.0000, A 0.000, B 0.000, C 0.000 }
gfCNCPoint2[13879] = {X 355.1421, Y 103.4631, Z -3.0000, A 0.000, B 0.000, C 0.000 }
gfCNCPoint2[13880] = {X 361.3005, Y 103.1290, Z -3.0000, A 0.000, B 0.000, C 0.000 }
gfCNCPoint2[13881] = {X 365.1928, Y 102.7584, Z -3.0000, A 0.000, B 0.000, C 0.000 }
gfCNCPoint2[13882] = {X 369.0628, Y 102.2011, Z -3.0000, A 0.000, B 0.000, C 0.000 }
gfCNCPoint2[13883] = {X 372.9015, Y 101.4583, Z -3.0000, A 0.000, B 0.000, C 0.000 }
gfCNCPoint2[13884] = {X 375.2297, Y 100.8563, Z -3.0000, A 0.000, B 0.000, C 0.000 }
gfCNCPoint2[13885] = {X 377.5107, Y 100.0950, Z -3.0000, A 0.000, B 0.000, C 0.000 }
gfCNCPoint2[13886] = {X 391.9985, Y 100.0950, Z -3.0000, A 0.000, B 0.000, C 0.000 }
gfCNCPoint2[13887] = {X 392.4673, Y 100.8812, Z -3.0000, A 0.000, B 0.000, C 0.000 }
gfCNCPoint2[13888] = {X 393.0746, Y 101.5660, Z -3.0000, A 0.000, B 0.000, C 0.000 }
gfCNCPoint2[13889] = {X 393.7991, Y 102.1254, Z -3.0000, A 0.000, B 0.000, C 0.000 }
gfCNCPoint2[13890] = {X 394.6154, Y 102.5396, Z -3.0000, A 0.000, B 0.000, C 0.000 }
gfCNCPoint2[13891] = {X 395.4946, Y 102.7942, Z -3.0000, A 0.000, B 0.000, C 0.000 }
gfCNCPoint2[13892] = {X 396.4059, Y 102.8800, Z -3.0000, A 0.000, B 0.000, C 0.000 }
gfCNCPoint2[13893] = {X 415.7067, Y 102.8800, Z -3.0000, A 0.000, B 0.000, C 0.000 }
gfCNCPoint2[13894] = {X 416.6180, Y 102.7942, Z -3.0000, A 0.000, B 0.000, C 0.000 }
gfCNCPoint2[13895] = {X 417.4973, Y 102.5396, Z -3.0000, A 0.000, B 0.000, C 0.000 }
gfCNCPoint2[13896] = {X 418.3135, Y 102.1254, Z -3.0000, A 0.000, B 0.000, C 0.000 }
gfCNCPoint2[13897] = {X 419.0381, Y 101.5660, Z -3.0000, A 0.000, B 0.000, C 0.000 }
gfCNCPoint2[13898] = {X 419.6454, Y 100.8812, Z -3.0000, A 0.000, B 0.000, C 0.000 }
gfCNCPoint2[13899] = {X 420.1141, Y 100.0950, Z -3.0000, A 0.000, B 0.000, C 0.000 }
gfCNCPoint2[13900] = {X 443.7019, Y 100.0950, Z -3.0000, A 0.000, B 0.000, C 0.000 }
gfCNCPoint2[13901] = {X 443.7019, Y 90.4950, Z -3.0000, A 0.000, B 0.000, C 0.000 }
gfCNCPoint2[13902] = {X 448.3231, Y 90.4950, Z -3.0000, A 0.000, B 0.000, C 0.000 }
gfCNCPoint2[13903] = {X 448.4021, Y 90.3747, Z -3.0000, A 0.000, B 0.000, C 0.000 }
gfCNCPoint2[13904] = {X 448.4825, Y 90.2554, Z -3.0000, A 0.000, B 0.000, C 0.000 }
gfCNCPoint2[13905] = {X 445.7346, Y 89.1782, Z -3.0000, A 0.000, B 0.000, C 0.000 }
gfCNCPoint2[13906] = {X 443.7019, Y 90.4950, Z -3.0000, A 0.000, B 0.000, C 0.000 }
gfCNCPoint2[13907] = {X 443.7019, Y 92.8950, Z -3.0000, A 0.000, B 0.000, C 0.000 }
gfCNCPoint2[13908] = {X 449.7243, Y 92.8950, Z -3.0000, A 0.000, B 0.000, C 0.000 }
gfCNCPoint2[13909] = {X 450.0698, Y 92.2375, Z -3.0000, A 0.000, B 0.000, C 0.000 }
gfCNCPoint2[13910] = {X 450.4647, Y 91.6084, Z -3.0000, A 0.000, B 0.000, C 0.000 }
gfCNCPoint2[13911] = {X 451.3969, Y 90.4463, Z -3.0000, A 0.000, B 0.000, C 0.000 }
gfCNCPoint2[13912] = {X 452.4963, Y 89.4409, Z -3.0000, A 0.000, B 0.000, C 0.000 }
gfCNCPoint2[13913] = {X 452.4963, Y 89.2510, Z -3.0000, A 0.000, B 0.000, C 0.000 }
gfCNCPoint2[13914] = {X 445.4636, Y 86.4941, Z -3.0000, A 0.000, B 0.000, C 0.000 }
gfCNCPoint2[13915] = {X 435.5827, Y 92.8950, Z -3.0000, A 0.000, B 0.000, C 0.000 }
gfCNCPoint2[13916] = {X 443.7019, Y 92.8950, Z -3.0000, A 0.000, B 0.000, C 0.000 }
gfCNCPoint2[13917] = {X 443.7019, Y 95.2950, Z -3.0000, A 0.000, B 0.000, C 0.000 }
gfCNCPoint2[13918] = {X 451.3983, Y 95.2950, Z -3.0000, A 0.000, B 0.000, C 0.000 }
gfCNCPoint2[13919] = {X 451.7785, Y 94.1744, Z -3.0000, A 0.000, B 0.000, C 0.000 }
gfCNCPoint2[13920] = {X 452.3352, Y 93.1303, Z -3.0000, A 0.000, B 0.000, C 0.000 }
gfCNCPoint2[13921] = {X 453.0536, Y 92.1901, Z -3.0000, A 0.000, B 0.000, C 0.000 }
gfCNCPoint2[13922] = {X 453.9149, Y 91.3787, Z -3.0000, A 0.000, B 0.000, C 0.000 }
gfCNCPoint2[13923] = {X 454.8963, Y 90.7176, Z -3.0000, A 0.000, B 0.000, C 0.000 }
gfCNCPoint2[13924] = {X 454.8963, Y 87.6139, Z -3.0000, A 0.000, B 0.000, C 0.000 }
gfCNCPoint2[13925] = {X 445.1927, Y 83.8101, Z -3.0000, A 0.000, B 0.000, C 0.000 }
gfCNCPoint2[13926] = {X 427.4635, Y 95.2950, Z -3.0000, A 0.000, B 0.000, C 0.000 }
gfCNCPoint2[13927] = {X 443.7019, Y 95.2950, Z -3.0000, A 0.000, B 0.000, C 0.000 }
gfCNCPoint2[13928] = {X 443.7019, Y 97.6950, Z -3.0000, A 0.000, B 0.000, C 0.000 }
gfCNCPoint2[13929] = {X 453.5796, Y 97.6950, Z -3.0000, A 0.000, B 0.000, C 0.000 }
gfCNCPoint2[13930] = {X 453.5796, Y 97.0659, Z -3.0000, A 0.000, B 0.000, C 0.000 }
gfCNCPoint2[13931] = {X 453.6990, Y 95.9930, Z -3.0000, A 0.000, B 0.000, C 0.000 }
gfCNCPoint2[13932] = {X 454.0514, Y 94.9725, Z -3.0000, A 0.000, B 0.000, C 0.000 }
gfCNCPoint2[13933] = {X 454.6196, Y 94.0545, Z -3.0000, A 0.000, B 0.000, C 0.000 }
gfCNCPoint2[13934] = {X 455.3757, Y 93.2839, Z -3.0000, A 0.000, B 0.000, C 0.000 }
gfCNCPoint2[13935] = {X 456.2827, Y 92.6984, Z -3.0000, A 0.000, B 0.000, C 0.000 }
gfCNCPoint2[13936] = {X 457.2963, Y 92.3266, Z -3.0000, A 0.000, B 0.000, C 0.000 }
gfCNCPoint2[13937] = {X 457.2963, Y 85.9769, Z -3.0000, A 0.000, B 0.000, C 0.000 }
gfCNCPoint2[13938] = {X 444.9217, Y 81.1261, Z -3.0000, A 0.000, B 0.000, C 0.000 }
gfCNCPoint2[13939] = {X 420.5854, Y 96.8910, Z -3.0000, A 0.000, B 0.000, C 0.000 }
gfCNCPoint2[13940] = {X 420.5867, Y 97.0659, Z -3.0000, A 0.000, B 0.000, C 0.000 }
gfCNCPoint2[13941] = {X 420.5867, Y 97.6950, Z -3.0000, A 0.000, B 0.000, C 0.000 }
gfCNCPoint2[13942] = {X 443.7019, Y 97.6950, Z -3.0000, A 0.000, B 0.000, C 0.000 }
gfCNCPoint2[13943] = {X 443.7019, Y 100.0950, Z -3.0000, A 0.000, B 0.000, C 0.000 }
gfCNCPoint2[13944] = {X 454.0522, Y 100.0950, Z -3.0000, A 0.000, B 0.000, C 0.000 }
gfCNCPoint2[13945] = {X 454.5209, Y 100.8812, Z -3.0000, A 0.000, B 0.000, C 0.000 }
gfCNCPoint2[13946] = {X 455.1282, Y 101.5660, Z -3.0000, A 0.000, B 0.000, C 0.000 }
gfCNCPoint2[13947] = {X 455.8528, Y 102.1254, Z -3.0000, A 0.000, B 0.000, C 0.000 }
gfCNCPoint2[13948] = {X 456.6690, Y 102.5396, Z -3.0000, A 0.000, B 0.000, C 0.000 }
gfCNCPoint2[13949] = {X 457.5483, Y 102.7942, Z -3.0000, A 0.000, B 0.000, C 0.000 }
gfCNCPoint2[13950] = {X 458.4596, Y 102.8800, Z -3.0000, A 0.000, B 0.000, C 0.000 }
gfCNCPoint2[13951] = {X 475.0000, Y 102.8800, Z -3.0000, A 0.000, B 0.000, C 0.000 }
gfCNCPoint2[13952] = {X 475.9113, Y 102.7942, Z -3.0000, A 0.000, B 0.000, C 0.000 }
gfCNCPoint2[13953] = {X 476.7906, Y 102.5396, Z -3.0000, A 0.000, B 0.000, C 0.000 }
gfCNCPoint2[13954] = {X 477.6068, Y 102.1254, Z -3.0000, A 0.000, B 0.000, C 0.000 }
gfCNCPoint2[13955] = {X 478.3314, Y 101.5660, Z -3.0000, A 0.000, B 0.000, C 0.000 }
gfCNCPoint2[13956] = {X 478.9387, Y 100.8812, Z -3.0000, A 0.000, B 0.000, C 0.000 }
gfCNCPoint2[13957] = {X 479.4074, Y 100.0950, Z -3.0000, A 0.000, B 0.000, C 0.000 }
gfCNCPoint2[13958] = {X 507.6818, Y 100.0950, Z -3.0000, A 0.000, B 0.000, C 0.000 }
gfCNCPoint2[13959] = {X 507.6818, Y 107.6950, Z -3.0000, A 0.000, B 0.000, C 0.000 }
gfCNCPoint2[13960] = {X 507.6818, Y 107.6950, Z 0.0000, A 0.000, B 0.000, C 0.000 }
gfCNCPoint2[13961] = {X 507.6818, Y 107.6950, Z 11.0000, A 0.000, B 0.000, C 0.000 }
gfCNCPoint2[13962] = {X 108.5558, Y 40.9003, Z 11.0000, A 0.000, B 0.000, C 0.000 }
gfCNCPoint2[13963] = {X 108.5558, Y 40.9003, Z 0.8333, A 0.000, B 0.000, C 0.000 }
gfCNCPoint2[13964] = {X 108.5558, Y 40.9003, Z -3.0000, A 0.000, B 0.000, C 0.000 }
gfCNCPoint2[13965] = {X 108.0651, Y 42.0994, Z -3.0000, A 0.000, B 0.000, C 0.000 }
gfCNCPoint2[13966] = {X 108.0933, Y 42.0503, Z -3.0000, A 0.000, B 0.000, C 0.000 }
gfCNCPoint2[13967] = {X 108.1221, Y 42.0015, Z -3.0000, A 0.000, B 0.000, C 0.000 }
gfCNCPoint2[13968] = {X 108.5470, Y 41.3856, Z -3.0000, A 0.000, B 0.000, C 0.000 }
gfCNCPoint2[13969] = {X 109.0466, Y 40.8285, Z -3.0000, A 0.000, B 0.000, C 0.000 }
gfCNCPoint2[13970] = {X 109.0465, Y 39.7012, Z -3.0000, A 0.000, B 0.000, C 0.000 }
gfCNCPoint2[13971] = {X 108.5558, Y 40.9003, Z -3.0000, A 0.000, B 0.000, C 0.000 }
gfCNCPoint2[13972] = {X 108.5558, Y 40.9003, Z 0.0000, A 0.000, B 0.000, C 0.000 }
gfCNCPoint2[13973] = {X 108.5558, Y 40.9003, Z 11.0000, A 0.000, B 0.000, C 0.000 }
gfCNCPoint2[13974] = {X 95.6839, Y 40.8752, Z 11.0000, A 0.000, B 0.000, C 0.000 }
gfCNCPoint2[13975] = {X 95.6839, Y 40.8752, Z 0.8333, A 0.000, B 0.000, C 0.000 }
gfCNCPoint2[13976] = {X 95.6839, Y 40.8752, Z -3.0000, A 0.000, B 0.000, C 0.000 }
gfCNCPoint2[13977] = {X 95.2104, Y 39.7173, Z -3.0000, A 0.000, B 0.000, C 0.000 }
gfCNCPoint2[13978] = {X 95.2105, Y 40.8689, Z -3.0000, A 0.000, B 0.000, C 0.000 }
gfCNCPoint2[13979] = {X 95.7330, Y 41.4112, Z -3.0000, A 0.000, B 0.000, C 0.000 }
gfCNCPoint2[13980] = {X 96.1574, Y 42.0332, Z -3.0000, A 0.000, B 0.000, C 0.000 }
gfCNCPoint2[13981] = {X 95.6839, Y 40.8752, Z -3.0000, A 0.000, B 0.000, C 0.000 }
gfCNCPoint2[13982] = {X 95.6839, Y 40.8752, Z 0.0000, A 0.000, B 0.000, C 0.000 }
gfCNCPoint2[13983] = {X 95.6839, Y 40.8752, Z 11.0000, A 0.000, B 0.000, C 0.000 }
gfCNCPoint2[13984] = {X -7.6965, Y 43.1529, Z 11.0000, A 0.000, B 0.000, C 0.000 }
gfCNCPoint2[13985] = {X -7.6965, Y 43.1529, Z 0.0000, A 0.000, B 0.000, C 0.000 }
gfCNCPoint2[13986] = {X -7.6965, Y 43.1529, Z -3.0000, A 0.000, B 0.000, C 0.000 }
gfCNCPoint2[13987] = {X -3.6965, Y 30.8010, Z -3.0000, A 0.000, B 0.000, C 0.000 }
gfCNCPoint2[13988] = {X -3.3664, Y 29.8867, Z -3.0000, A 0.000, B 0.000, C 0.000 }
gfCNCPoint2[13989] = {X -2.9761, Y 28.9965, Z -3.0000, A 0.000, B 0.000, C 0.000 }
gfCNCPoint2[13990] = {X -2.3495, Y 27.8700, Z -3.0000, A 0.000, B 0.000, C 0.000 }
gfCNCPoint2[13991] = {X -1.5932, Y 26.8262, Z -3.0000, A 0.000, B 0.000, C 0.000 }
gfCNCPoint2[13992] = {X -0.7179, Y 25.8800, Z -3.0000, A 0.000, B 0.000, C 0.000 }
gfCNCPoint2[13993] = {X 0.2640, Y 25.0449, Z -3.0000, A 0.000, B 0.000, C 0.000 }
gfCNCPoint2[13994] = {X 1.3384, Y 24.3328, Z -3.0000, A 0.000, B 0.000, C 0.000 }
gfCNCPoint2[13995] = {X 0.5785, Y 23.9224, Z -3.0000, A 0.000, B 0.000, C 0.000 }
gfCNCPoint2[13996] = {X -0.0866, Y 23.3716, Z -3.0000, A 0.000, B 0.000, C 0.000 }
gfCNCPoint2[13997] = {X -0.6312, Y 22.7015, Z -3.0000, A 0.000, B 0.000, C 0.000 }
gfCNCPoint2[13998] = {X -1.0345, Y 21.9378, Z -3.0000, A 0.000, B 0.000, C 0.000 }
gfCNCPoint2[13999] = {X -3.6458, Y 15.5423, Z -3.0000, A 0.000, B 0.000, C 0.000 }
gfCNCPoint2[14000] = {X -3.6717, Y 15.4774, Z -3.0000, A 0.000, B 0.000, C 0.000 }
gfCNCPoint2[14001] = {X -3.6965, Y 15.4121, Z -3.0000, A 0.000, B 0.000, C 0.000 }
gfCNCPoint2[14002] = {X -7.6965, Y 4.6510, Z -3.0000, A 0.000, B 0.000, C 0.000 }
gfCNCPoint2[14003] = {X -7.6965, Y 4.6510, Z 0.0000, A 0.000, B 0.000, C 0.000 }
gfCNCPoint2[14004] = {X -7.6965, Y 4.6510, Z 11.0000, A 0.000, B 0.000, C 0.000 }
gfCNCPoint2[14005] = {X -7.6965, Y 16.4124, Z 11.0000, A 0.000, B 0.000, C 0.000 }
gfCNCPoint2[14006] = {X -7.6965, Y 16.4124, Z 0.0000, A 0.000, B 0.000, C 0.000 }
gfCNCPoint2[14007] = {X -7.6965, Y 16.4124, Z -3.0000, A 0.000, B 0.000, C 0.000 }
gfCNCPoint2[14008] = {X -4.8868, Y 16.4124, Z -3.0000, A 0.000, B 0.000, C 0.000 }
gfCNCPoint2[14009] = {X -3.6965, Y 12.5936, Z -3.0000, A 0.000, B 0.000, C 0.000 }
gfCNCPoint2[14010] = {X -3.6605, Y 12.4833, Z -3.0000, A 0.000, B 0.000, C 0.000 }
gfCNCPoint2[14011] = {X -3.6215, Y 12.3740, Z -3.0000, A 0.000, B 0.000, C 0.000 }
gfCNCPoint2[14012] = {X -3.1666, Y 11.4827, Z -3.0000, A 0.000, B 0.000, C 0.000 }
gfCNCPoint2[14013] = {X -2.5188, Y 10.7200, Z -3.0000, A 0.000, B 0.000, C 0.000 }
gfCNCPoint2[14014] = {X -1.7129, Y 10.1268, Z -3.0000, A 0.000, B 0.000, C 0.000 }
gfCNCPoint2[14015] = {X -1.1157, Y 9.7861, Z -3.0000, A 0.000, B 0.000, C 0.000 }
gfCNCPoint2[14016] = {X -0.2292, Y 9.4045, Z -3.0000, A 0.000, B 0.000, C 0.000 }
gfCNCPoint2[14017] = {X 0.7198, Y 9.2292, Z -3.0000, A 0.000, B 0.000, C 0.000 }
gfCNCPoint2[14018] = {X 1.6841, Y 9.2690, Z -3.0000, A 0.000, B 0.000, C 0.000 }
gfCNCPoint2[14019] = {X 2.6154, Y 9.5219, Z -3.0000, A 0.000, B 0.000, C 0.000 }
gfCNCPoint2[14020] = {X 3.3921, Y 9.1587, Z -3.0000, A 0.000, B 0.000, C 0.000 }
gfCNCPoint2[14021] = {X 4.1906, Y 8.8464, Z -3.0000, A 0.000, B 0.000, C 0.000 }
gfCNCPoint2[14022] = {X 6.1023, Y 8.1768, Z -3.0000, A 0.000, B 0.000, C 0.000 }
gfCNCPoint2[14023] = {X 8.0646, Y 7.6746, Z -3.0000, A 0.000, B 0.000, C 0.000 }
gfCNCPoint2[14024] = {X 10.0629, Y 7.3436, Z -3.0000, A 0.000, B 0.000, C 0.000 }
gfCNCPoint2[14025] = {X 12.0824, Y 7.1863, Z -3.0000, A 0.000, B 0.000, C 0.000 }
gfCNCPoint2[14026] = {X 14.1079, Y 7.2039, Z -3.0000, A 0.000, B 0.000, C 0.000 }
gfCNCPoint2[14027] = {X 16.1243, Y 7.3961, Z -3.0000, A 0.000, B 0.000, C 0.000 }
gfCNCPoint2[14028] = {X 17.9475, Y 7.7297, Z -3.0000, A 0.000, B 0.000, C 0.000 }
gfCNCPoint2[14029] = {X 19.7250, Y 8.2548, Z -3.0000, A 0.000, B 0.000, C 0.000 }
gfCNCPoint2[14030] = {X 21.4369, Y 8.9654, Z -3.0000, A 0.000, B 0.000, C 0.000 }
gfCNCPoint2[14031] = {X 23.0638, Y 9.8534, Z -3.0000, A 0.000, B 0.000, C 0.000 }
gfCNCPoint2[14032] = {X 24.5873, Y 10.9090, Z -3.0000, A 0.000, B 0.000, C 0.000 }
gfCNCPoint2[14033] = {X 25.6725, Y 11.8577, Z -3.0000, A 0.000, B 0.000, C 0.000 }
gfCNCPoint2[14034] = {X 26.6459, Y 12.9208, Z -3.0000, A 0.000, B 0.000, C 0.000 }
gfCNCPoint2[14035] = {X 27.4956, Y 14.0852, Z -3.0000, A 0.000, B 0.000, C 0.000 }
gfCNCPoint2[14036] = {X 28.2111, Y 15.3365, Z -3.0000, A 0.000, B 0.000, C 0.000 }
gfCNCPoint2[14037] = {X 28.7835, Y 16.6594, Z -3.0000, A 0.000, B 0.000, C 0.000 }
gfCNCPoint2[14038] = {X 29.2582, Y 18.3156, Z -3.0000, A 0.000, B 0.000, C 0.000 }
gfCNCPoint2[14039] = {X 29.5398, Y 20.0152, Z -3.0000, A 0.000, B 0.000, C 0.000 }
gfCNCPoint2[14040] = {X 29.6249, Y 21.7360, Z -3.0000, A 0.000, B 0.000, C 0.000 }
gfCNCPoint2[14041] = {X 29.5122, Y 23.4551, Z -3.0000, A 0.000, B 0.000, C 0.000 }
gfCNCPoint2[14042] = {X 29.2032, Y 25.1501, Z -3.0000, A 0.000, B 0.000, C 0.000 }
gfCNCPoint2[14043] = {X 28.7612, Y 26.5965, Z -3.0000, A 0.000, B 0.000, C 0.000 }
gfCNCPoint2[14044] = {X 28.1360, Y 27.9737, Z -3.0000, A 0.000, B 0.000, C 0.000 }
gfCNCPoint2[14045] = {X 27.3383, Y 29.2586, Z -3.0000, A 0.000, B 0.000, C 0.000 }
gfCNCPoint2[14046] = {X 26.3813, Y 30.4298, Z -3.0000, A 0.000, B 0.000, C 0.000 }
gfCNCPoint2[14047] = {X 25.2811, Y 31.4676, Z -3.0000, A 0.000, B 0.000, C 0.000 }
gfCNCPoint2[14048] = {X 26.0851, Y 31.8097, Z -3.0000, A 0.000, B 0.000, C 0.000 }
gfCNCPoint2[14049] = {X 26.8039, Y 32.3067, Z -3.0000, A 0.000, B 0.000, C 0.000 }
gfCNCPoint2[14050] = {X 27.4079, Y 32.9381, Z -3.0000, A 0.000, B 0.000, C 0.000 }
gfCNCPoint2[14051] = {X 27.8726, Y 33.6781, Z -3.0000, A 0.000, B 0.000, C 0.000 }
gfCNCPoint2[14052] = {X 30.9100, Y 39.9530, Z -3.0000, A 0.000, B 0.000, C 0.000 }
gfCNCPoint2[14053] = {X 31.2306, Y 40.8622, Z -3.0000, A 0.000, B 0.000, C 0.000 }
gfCNCPoint2[14054] = {X 31.3415, Y 41.8197, Z -3.0000, A 0.000, B 0.000, C 0.000 }
gfCNCPoint2[14055] = {X 31.2374, Y 42.7781, Z -3.0000, A 0.000, B 0.000, C 0.000 }
gfCNCPoint2[14056] = {X 30.9234, Y 43.6895, Z -3.0000, A 0.000, B 0.000, C 0.000 }
gfCNCPoint2[14057] = {X 30.4150, Y 44.5085, Z -3.0000, A 0.000, B 0.000, C 0.000 }
gfCNCPoint2[14058] = {X 29.7377, Y 45.1945, Z -3.0000, A 0.000, B 0.000, C 0.000 }
gfCNCPoint2[14059] = {X 29.2014, Y 45.6281, Z -3.0000, A 0.000, B 0.000, C 0.000 }
gfCNCPoint2[14060] = {X 28.4969, Y 46.0912, Z -3.0000, A 0.000, B 0.000, C 0.000 }
gfCNCPoint2[14061] = {X 27.7160, Y 46.4093, Z -3.0000, A 0.000, B 0.000, C 0.000 }
gfCNCPoint2[14062] = {X 26.8884, Y 46.5702, Z -3.0000, A 0.000, B 0.000, C 0.000 }
gfCNCPoint2[14063] = {X 26.0453, Y 46.5679, Z -3.0000, A 0.000, B 0.000, C 0.000 }
gfCNCPoint2[14064] = {X 25.2185, Y 46.4026, Z -3.0000, A 0.000, B 0.000, C 0.000 }
gfCNCPoint2[14065] = {X 23.6418, Y 47.2470, Z -3.0000, A 0.000, B 0.000, C 0.000 }
gfCNCPoint2[14066] = {X 22.0144, Y 47.9889, Z -3.0000, A 0.000, B 0.000, C 0.000 }
gfCNCPoint2[14067] = {X 20.3429, Y 48.6254, Z -3.0000, A 0.000, B 0.000, C 0.000 }
gfCNCPoint2[14068] = {X 18.4181, Y 49.2355, Z -3.0000, A 0.000, B 0.000, C 0.000 }
gfCNCPoint2[14069] = {X 16.4468, Y 49.6730, Z -3.0000, A 0.000, B 0.000, C 0.000 }
gfCNCPoint2[14070] = {X 14.4446, Y 49.9346, Z -3.0000, A 0.000, B 0.000, C 0.000 }
gfCNCPoint2[14071] = {X 12.4271, Y 50.0181, Z -3.0000, A 0.000, B 0.000, C 0.000 }
gfCNCPoint2[14072] = {X 10.4102, Y 49.9230, Z -3.0000, A 0.000, B 0.000, C 0.000 }
gfCNCPoint2[14073] = {X 8.4095, Y 49.6499, Z -3.0000, A 0.000, B 0.000, C 0.000 }
gfCNCPoint2[14074] = {X 6.5320, Y 49.2143, Z -3.0000, A 0.000, B 0.000, C 0.000 }
gfCNCPoint2[14075] = {X 4.7153, Y 48.5707, Z -3.0000, A 0.000, B 0.000, C 0.000 }
gfCNCPoint2[14076] = {X 2.9824, Y 47.7272, Z -3.0000, A 0.000, B 0.000, C 0.000 }
gfCNCPoint2[14077] = {X 1.3551, Y 46.6945, Z -3.0000, A 0.000, B 0.000, C 0.000 }
gfCNCPoint2[14078] = {X 0.0297, Y 45.6276, Z -3.0000, A 0.000, B 0.000, C 0.000 }
gfCNCPoint2[14079] = {X -1.1484, Y 44.4002, Z -3.0000, A 0.000, B 0.000, C 0.000 }
gfCNCPoint2[14080] = {X -2.1600, Y 43.0322, Z -3.0000, A 0.000, B 0.000, C 0.000 }
gfCNCPoint2[14081] = {X -2.9886, Y 41.5462, Z -3.0000, A 0.000, B 0.000, C 0.000 }
gfCNCPoint2[14082] = {X -3.6205, Y 39.9666, Z -3.0000, A 0.000, B 0.000, C 0.000 }
gfCNCPoint2[14083] = {X -3.6591, Y 39.8468, Z -3.0000, A 0.000, B 0.000, C 0.000 }
gfCNCPoint2[14084] = {X -3.6965, Y 39.7267, Z -3.0000, A 0.000, B 0.000, C 0.000 }
gfCNCPoint2[14085] = {X -4.8691, Y 35.9025, Z -3.0000, A 0.000, B 0.000, C 0.000 }
gfCNCPoint2[14086] = {X -7.9909, Y 36.0289, Z -3.0000, A 0.000, B 0.000, C 0.000 }
gfCNCPoint2[14087] = {X -7.9909, Y 36.0289, Z 0.0000, A 0.000, B 0.000, C 0.000 }
gfCNCPoint2[14088] = {X -7.9909, Y 36.0289, Z 11.0000, A 0.000, B 0.000, C 0.000 }
gfCNCPoint2[14089] = {X 608.0000, Y 40.1201, Z 11.0000, A 0.000, B 0.000, C 0.000 }
gfCNCPoint2[14090] = {X 608.0000, Y 40.1201, Z 0.0000, A 0.000, B 0.000, C 0.000 }
gfCNCPoint2[14091] = {X 608.0000, Y 40.1201, Z -3.0000, A 0.000, B 0.000, C 0.000 }
gfCNCPoint2[14092] = {X 603.6965, Y 47.2357, Z -3.0000, A 0.000, B 0.000, C 0.000 }
gfCNCPoint2[14093] = {X 603.6633, Y 47.2897, Z -3.0000, A 0.000, B 0.000, C 0.000 }
gfCNCPoint2[14094] = {X 603.6293, Y 47.3432, Z -3.0000, A 0.000, B 0.000, C 0.000 }
gfCNCPoint2[14095] = {X 603.0930, Y 48.0160, Z -3.0000, A 0.000, B 0.000, C 0.000 }
gfCNCPoint2[14096] = {X 602.4339, Y 48.5691, Z -3.0000, A 0.000, B 0.000, C 0.000 }
gfCNCPoint2[14097] = {X 601.6783, Y 48.9807, Z -3.0000, A 0.000, B 0.000, C 0.000 }
gfCNCPoint2[14098] = {X 600.8561, Y 49.2343, Z -3.0000, A 0.000, B 0.000, C 0.000 }
gfCNCPoint2[14099] = {X 600.0000, Y 49.3200, Z -3.0000, A 0.000, B 0.000, C 0.000 }
gfCNCPoint2[14100] = {X 593.5565, Y 49.3200, Z -3.0000, A 0.000, B 0.000, C 0.000 }
gfCNCPoint2[14101] = {X 592.5952, Y 49.2117, Z -3.0000, A 0.000, B 0.000, C 0.000 }
gfCNCPoint2[14102] = {X 591.6822, Y 48.8922, Z -3.0000, A 0.000, B 0.000, C 0.000 }
gfCNCPoint2[14103] = {X 590.8631, Y 48.3775, Z -3.0000, A 0.000, B 0.000, C 0.000 }
gfCNCPoint2[14104] = {X 590.1790, Y 47.6935, Z -3.0000, A 0.000, B 0.000, C 0.000 }
gfCNCPoint2[14105] = {X 589.6643, Y 46.8744, Z -3.0000, A 0.000, B 0.000, C 0.000 }
gfCNCPoint2[14106] = {X 589.3448, Y 45.9613, Z -3.0000, A 0.000, B 0.000, C 0.000 }
gfCNCPoint2[14107] = {X 589.2365, Y 45.0000, Z -3.0000, A 0.000, B 0.000, C 0.000 }
gfCNCPoint2[14108] = {X 589.2365, Y 44.0644, Z -3.0000, A 0.000, B 0.000, C 0.000 }
gfCNCPoint2[14109] = {X 589.3412, Y 43.1363, Z -3.0000, A 0.000, B 0.000, C 0.000 }
gfCNCPoint2[14110] = {X 589.6410, Y 42.2517, Z -3.0000, A 0.000, B 0.000, C 0.000 }
gfCNCPoint2[14111] = {X 590.1222, Y 41.4512, Z -3.0000, A 0.000, B 0.000, C 0.000 }
gfCNCPoint2[14112] = {X 590.7628, Y 40.7715, Z -3.0000, A 0.000, B 0.000, C 0.000 }
gfCNCPoint2[14113] = {X 590.7632, Y 33.5299, Z -3.0000, A 0.000, B 0.000, C 0.000 }
gfCNCPoint2[14114] = {X 585.4453, Y 46.6524, Z -3.0000, A 0.000, B 0.000, C 0.000 }
gfCNCPoint2[14115] = {X 585.0755, Y 47.3550, Z -3.0000, A 0.000, B 0.000, C 0.000 }
gfCNCPoint2[14116] = {X 584.5834, Y 47.9780, Z -3.0000, A 0.000, B 0.000, C 0.000 }
gfCNCPoint2[14117] = {X 583.9856, Y 48.5004, Z -3.0000, A 0.000, B 0.000, C 0.000 }
gfCNCPoint2[14118] = {X 583.3023, Y 48.9046, Z -3.0000, A 0.000, B 0.000, C 0.000 }
gfCNCPoint2[14119] = {X 582.3585, Y 49.2242, Z -3.0000, A 0.000, B 0.000, C 0.000 }
gfCNCPoint2[14120] = {X 581.3666, Y 49.3191, Z -3.0000, A 0.000, B 0.000, C 0.000 }
gfCNCPoint2[14121] = {X 580.3794, Y 49.1842, Z -3.0000, A 0.000, B 0.000, C 0.000 }
gfCNCPoint2[14122] = {X 579.4493, Y 48.8268, Z -3.0000, A 0.000, B 0.000, C 0.000 }
gfCNCPoint2[14123] = {X 578.6259, Y 48.2657, Z -3.0000, A 0.000, B 0.000, C 0.000 }
gfCNCPoint2[14124] = {X 577.9529, Y 47.5309, Z -3.0000, A 0.000, B 0.000, C 0.000 }
gfCNCPoint2[14125] = {X 577.4662, Y 46.6615, Z -3.0000, A 0.000, B 0.000, C 0.000 }
gfCNCPoint2[14126] = {X 572.0182, Y 33.3399, Z -3.0000, A 0.000, B 0.000, C 0.000 }
gfCNCPoint2[14127] = {X 572.0215, Y 40.7720, Z -3.0000, A 0.000, B 0.000, C 0.000 }
gfCNCPoint2[14128] = {X 572.6589, Y 41.4429, Z -3.0000, A 0.000, B 0.000, C 0.000 }
gfCNCPoint2[14129] = {X 573.1389, Y 42.2342, Z -3.0000, A 0.000, B 0.000, C 0.000 }
gfCNCPoint2[14130] = {X 573.4392, Y 43.1095, Z -3.0000, A 0.000, B 0.000, C 0.000 }
gfCNCPoint2[14131] = {X 573.5463, Y 44.0287, Z -3.0000, A 0.000, B 0.000, C 0.000 }
gfCNCPoint2[14132] = {X 573.5464, Y 45.0000, Z -3.0000, A 0.000, B 0.000, C 0.000 }
gfCNCPoint2[14133] = {X 573.4381, Y 45.9613, Z -3.0000, A 0.000, B 0.000, C 0.000 }
gfCNCPoint2[14134] = {X 573.1186, Y 46.8744, Z -3.0000, A 0.000, B 0.000, C 0.000 }
gfCNCPoint2[14135] = {X 572.6039, Y 47.6935, Z -3.0000, A 0.000, B 0.000, C 0.000 }
gfCNCPoint2[14136] = {X 571.9199, Y 48.3775, Z -3.0000, A 0.000, B 0.000, C 0.000 }
gfCNCPoint2[14137] = {X 571.1008, Y 48.8922, Z -3.0000, A 0.000, B 0.000, C 0.000 }
gfCNCPoint2[14138] = {X 570.1877, Y 49.2117, Z -3.0000, A 0.000, B 0.000, C 0.000 }
gfCNCPoint2[14139] = {X 569.2264, Y 49.3200, Z -3.0000, A 0.000, B 0.000, C 0.000 }
gfCNCPoint2[14140] = {X 562.4443, Y 49.3200, Z -3.0000, A 0.000, B 0.000, C 0.000 }
gfCNCPoint2[14141] = {X 561.4830, Y 49.2117, Z -3.0000, A 0.000, B 0.000, C 0.000 }
gfCNCPoint2[14142] = {X 560.5699, Y 48.8922, Z -3.0000, A 0.000, B 0.000, C 0.000 }
gfCNCPoint2[14143] = {X 559.7508, Y 48.3775, Z -3.0000, A 0.000, B 0.000, C 0.000 }
gfCNCPoint2[14144] = {X 559.0668, Y 47.6935, Z -3.0000, A 0.000, B 0.000, C 0.000 }
gfCNCPoint2[14145] = {X 558.5521, Y 46.8744, Z -3.0000, A 0.000, B 0.000, C 0.000 }
gfCNCPoint2[14146] = {X 558.2326, Y 45.9613, Z -3.0000, A 0.000, B 0.000, C 0.000 }
gfCNCPoint2[14147] = {X 558.1243, Y 45.0000, Z -3.0000, A 0.000, B 0.000, C 0.000 }
gfCNCPoint2[14148] = {X 558.1243, Y 44.0645, Z -3.0000, A 0.000, B 0.000, C 0.000 }
gfCNCPoint2[14149] = {X 558.2288, Y 43.1360, Z -3.0000, A 0.000, B 0.000, C 0.000 }
gfCNCPoint2[14150] = {X 558.5289, Y 42.2511, Z -3.0000, A 0.000, B 0.000, C 0.000 }
gfCNCPoint2[14151] = {X 559.0108, Y 41.4505, Z -3.0000, A 0.000, B 0.000, C 0.000 }
gfCNCPoint2[14152] = {X 559.6524, Y 40.7712, Z -3.0000, A 0.000, B 0.000, C 0.000 }
gfCNCPoint2[14153] = {X 559.6524, Y 9.2307, Z -3.0000, A 0.000, B 0.000, C 0.000 }
gfCNCPoint2[14154] = {X 559.0138, Y 8.5597, Z -3.0000, A 0.000, B 0.000, C 0.000 }
gfCNCPoint2[14155] = {X 558.5329, Y 7.7679, Z -3.0000, A 0.000, B 0.000, C 0.000 }
gfCNCPoint2[14156] = {X 558.2318, Y 6.8919, Z -3.0000, A 0.000, B 0.000, C 0.000 }
gfCNCPoint2[14157] = {X 558.1245, Y 5.9718, Z -3.0000, A 0.000, B 0.000, C 0.000 }
gfCNCPoint2[14158] = {X 558.1243, Y 5.0000, Z -3.0000, A 0.000, B 0.000, C 0.000 }
gfCNCPoint2[14159] = {X 558.2326, Y 4.0387, Z -3.0000, A 0.000, B 0.000, C 0.000 }
gfCNCPoint2[14160] = {X 558.5521, Y 3.1256, Z -3.0000, A 0.000, B 0.000, C 0.000 }
gfCNCPoint2[14161] = {X 559.0668, Y 2.3065, Z -3.0000, A 0.000, B 0.000, C 0.000 }
gfCNCPoint2[14162] = {X 559.7508, Y 1.6225, Z -3.0000, A 0.000, B 0.000, C 0.000 }
gfCNCPoint2[14163] = {X 560.5699, Y 1.1078, Z -3.0000, A 0.000, B 0.000, C 0.000 }
gfCNCPoint2[14164] = {X 561.4830, Y 0.7883, Z -3.0000, A 0.000, B 0.000, C 0.000 }
gfCNCPoint2[14165] = {X 562.4443, Y 0.6800, Z -3.0000, A 0.000, B 0.000, C 0.000 }
gfCNCPoint2[14166] = {X 570.9376, Y 0.6800, Z -3.0000, A 0.000, B 0.000, C 0.000 }
gfCNCPoint2[14167] = {X 571.8988, Y 0.7883, Z -3.0000, A 0.000, B 0.000, C 0.000 }
gfCNCPoint2[14168] = {X 572.8119, Y 1.1078, Z -3.0000, A 0.000, B 0.000, C 0.000 }
gfCNCPoint2[14169] = {X 573.6310, Y 1.6225, Z -3.0000, A 0.000, B 0.000, C 0.000 }
gfCNCPoint2[14170] = {X 574.3151, Y 2.3065, Z -3.0000, A 0.000, B 0.000, C 0.000 }
gfCNCPoint2[14171] = {X 574.8297, Y 3.1256, Z -3.0000, A 0.000, B 0.000, C 0.000 }
gfCNCPoint2[14172] = {X 575.1492, Y 4.0387, Z -3.0000, A 0.000, B 0.000, C 0.000 }
gfCNCPoint2[14173] = {X 575.2576, Y 5.0000, Z -3.0000, A 0.000, B 0.000, C 0.000 }
gfCNCPoint2[14174] = {X 575.2576, Y 5.9342, Z -3.0000, A 0.000, B 0.000, C 0.000 }
gfCNCPoint2[14175] = {X 575.1835, Y 6.7307, Z -3.0000, A 0.000, B 0.000, C 0.000 }
gfCNCPoint2[14176] = {X 574.9638, Y 7.4998, Z -3.0000, A 0.000, B 0.000, C 0.000 }
gfCNCPoint2[14177] = {X 574.6061, Y 8.2153, Z -3.0000, A 0.000, B 0.000, C 0.000 }
gfCNCPoint2[14178] = {X 581.1909, Y 24.3706, Z -3.0000, A 0.000, B 0.000, C 0.000 }
gfCNCPoint2[14179] = {X 587.8459, Y 8.0944, Z -3.0000, A 0.000, B 0.000, C 0.000 }
gfCNCPoint2[14180] = {X 587.5317, Y 7.4232, Z -3.0000, A 0.000, B 0.000, C 0.000 }
gfCNCPoint2[14181] = {X 587.3369, Y 6.7083, Z -3.0000, A 0.000, B 0.000, C 0.000 }
gfCNCPoint2[14182] = {X 587.2671, Y 5.9705, Z -3.0000, A 0.000, B 0.000, C 0.000 }
gfCNCPoint2[14183] = {X 587.2670, Y 5.0000, Z -3.0000, A 0.000, B 0.000, C 0.000 }
gfCNCPoint2[14184] = {X 587.3753, Y 4.0387, Z -3.0000, A 0.000, B 0.000, C 0.000 }
gfCNCPoint2[14185] = {X 587.6948, Y 3.1256, Z -3.0000, A 0.000, B 0.000, C 0.000 }
gfCNCPoint2[14186] = {X 588.2094, Y 2.3065, Z -3.0000, A 0.000, B 0.000, C 0.000 }
gfCNCPoint2[14187] = {X 588.8935, Y 1.6225, Z -3.0000, A 0.000, B 0.000, C 0.000 }
gfCNCPoint2[14188] = {X 589.7126, Y 1.1078, Z -3.0000, A 0.000, B 0.000, C 0.000 }
gfCNCPoint2[14189] = {X 590.6257, Y 0.7883, Z -3.0000, A 0.000, B 0.000, C 0.000 }
gfCNCPoint2[14190] = {X 591.5870, Y 0.6800, Z -3.0000, A 0.000, B 0.000, C 0.000 }
gfCNCPoint2[14191] = {X 600.0000, Y 0.6800, Z -3.0000, A 0.000, B 0.000, C 0.000 }
gfCNCPoint2[14192] = {X 600.8561, Y 0.7657, Z -3.0000, A 0.000, B 0.000, C 0.000 }
gfCNCPoint2[14193] = {X 601.6783, Y 1.0193, Z -3.0000, A 0.000, B 0.000, C 0.000 }
gfCNCPoint2[14194] = {X 602.4339, Y 1.4309, Z -3.0000, A 0.000, B 0.000, C 0.000 }
gfCNCPoint2[14195] = {X 603.0930, Y 1.9840, Z -3.0000, A 0.000, B 0.000, C 0.000 }
gfCNCPoint2[14196] = {X 603.6293, Y 2.6568, Z -3.0000, A 0.000, B 0.000, C 0.000 }
gfCNCPoint2[14197] = {X 603.6633, Y 2.7103, Z -3.0000, A 0.000, B 0.000, C 0.000 }
gfCNCPoint2[14198] = {X 603.6965, Y 2.7643, Z -3.0000, A 0.000, B 0.000, C 0.000 }
gfCNCPoint2[14199] = {X 608.0000, Y 9.8799, Z -3.0000, A 0.000, B 0.000, C 0.000 }
gfCNCPoint2[14200] = {X 608.0000, Y 9.8799, Z 0.0000, A 0.000, B 0.000, C 0.000 }
gfCNCPoint2[14201] = {X 608.0000, Y 9.8799, Z 11.0000, A 0.000, B 0.000, C 0.000 }
gfCNCPoint2[14202] = {X -7.6965, Y 16.7862, Z 11.0000, A 0.000, B 0.000, C 0.000 }
gfCNCPoint2[14203] = {X -7.6965, Y 16.7862, Z 0.0000, A 0.000, B 0.000, C 0.000 }
gfCNCPoint2[14204] = {X -7.6965, Y 16.7862, Z -3.0000, A 0.000, B 0.000, C 0.000 }
gfCNCPoint2[14205] = {X -4.6246, Y 16.7862, Z -3.0000, A 0.000, B 0.000, C 0.000 }
gfCNCPoint2[14206] = {X -3.6965, Y 12.8954, Z -3.0000, A 0.000, B 0.000, C 0.000 }
gfCNCPoint2[14207] = {X -3.6290, Y 12.6463, Z -3.0000, A 0.000, B 0.000, C 0.000 }
gfCNCPoint2[14208] = {X -3.5465, Y 12.4018, Z -3.0000, A 0.000, B 0.000, C 0.000 }
gfCNCPoint2[14209] = {X -3.1000, Y 11.5271, Z -3.0000, A 0.000, B 0.000, C 0.000 }
gfCNCPoint2[14210] = {X -2.4643, Y 10.7785, Z -3.0000, A 0.000, B 0.000, C 0.000 }
gfCNCPoint2[14211] = {X -1.6733, Y 10.1963, Z -3.0000, A 0.000, B 0.000, C 0.000 }
gfCNCPoint2[14212] = {X -1.0760, Y 9.8556, Z -3.0000, A 0.000, B 0.000, C 0.000 }
gfCNCPoint2[14213] = {X -0.1974, Y 9.4785, Z -3.0000, A 0.000, B 0.000, C 0.000 }
gfCNCPoint2[14214] = {X 0.7434, Y 9.3078, Z -3.0000, A 0.000, B 0.000, C 0.000 }
gfCNCPoint2[14215] = {X 1.6985, Y 9.3523, Z -3.0000, A 0.000, B 0.000, C 0.000 }
gfCNCPoint2[14216] = {X 2.6194, Y 9.6097, Z -3.0000, A 0.000, B 0.000, C 0.000 }
gfCNCPoint2[14217] = {X 3.4077, Y 9.2390, Z -3.0000, A 0.000, B 0.000, C 0.000 }
gfCNCPoint2[14218] = {X 4.2188, Y 8.9213, Z -3.0000, A 0.000, B 0.000, C 0.000 }
gfCNCPoint2[14219] = {X 6.1242, Y 8.2537, Z -3.0000, A 0.000, B 0.000, C 0.000 }
gfCNCPoint2[14220] = {X 8.0801, Y 7.7531, Z -3.0000, A 0.000, B 0.000, C 0.000 }
gfCNCPoint2[14221] = {X 10.0720, Y 7.4231, Z -3.0000, A 0.000, B 0.000, C 0.000 }
gfCNCPoint2[14222] = {X 12.0849, Y 7.2663, Z -3.0000, A 0.000, B 0.000, C 0.000 }
gfCNCPoint2[14223] = {X 14.1038, Y 7.2837, Z -3.0000, A 0.000, B 0.000, C 0.000 }
gfCNCPoint2[14224] = {X 16.1137, Y 7.4754, Z -3.0000, A 0.000, B 0.000, C 0.000 }
gfCNCPoint2[14225] = {X 17.9286, Y 7.8075, Z -3.0000, A 0.000, B 0.000, C 0.000 }
gfCNCPoint2[14226] = {X 19.6981, Y 8.3301, Z -3.0000, A 0.000, B 0.000, C 0.000 }
gfCNCPoint2[14227] = {X 21.4022, Y 9.0374, Z -3.0000, A 0.000, B 0.000, C 0.000 }
gfCNCPoint2[14228] = {X 23.0217, Y 9.9215, Z -3.0000, A 0.000, B 0.000, C 0.000 }
gfCNCPoint2[14229] = {X 24.5383, Y 10.9722, Z -3.0000, A 0.000, B 0.000, C 0.000 }
gfCNCPoint2[14230] = {X 25.6168, Y 11.9151, Z -3.0000, A 0.000, B 0.000, C 0.000 }
gfCNCPoint2[14231] = {X 26.5842, Y 12.9716, Z -3.0000, A 0.000, B 0.000, C 0.000 }
gfCNCPoint2[14232] = {X 27.4285, Y 14.1288, Z -3.0000, A 0.000, B 0.000, C 0.000 }
gfCNCPoint2[14233] = {X 28.1396, Y 15.3724, Z -3.0000, A 0.000, B 0.000, C 0.000 }
gfCNCPoint2[14234] = {X 28.7085, Y 16.6870, Z -3.0000, A 0.000, B 0.000, C 0.000 }
gfCNCPoint2[14235] = {X 29.1804, Y 18.3342, Z -3.0000, A 0.000, B 0.000, C 0.000 }
gfCNCPoint2[14236] = {X 29.4604, Y 20.0246, Z -3.0000, A 0.000, B 0.000, C 0.000 }
gfCNCPoint2[14237] = {X 29.5449, Y 21.7360, Z -3.0000, A 0.000, B 0.000, C 0.000 }
gfCNCPoint2[14238] = {X 29.4327, Y 23.4458, Z -3.0000, A 0.000, B 0.000, C 0.000 }
gfCNCPoint2[14239] = {X 29.1254, Y 25.1315, Z -3.0000, A 0.000, B 0.000, C 0.000 }
gfCNCPoint2[14240] = {X 28.6756, Y 26.5964, Z -3.0000, A 0.000, B 0.000, C 0.000 }
gfCNCPoint2[14241] = {X 28.0368, Y 27.9893, Z -3.0000, A 0.000, B 0.000, C 0.000 }
gfCNCPoint2[14242] = {X 27.2201, Y 29.2859, Z -3.0000, A 0.000, B 0.000, C 0.000 }
gfCNCPoint2[14243] = {X 26.2396, Y 30.4636, Z -3.0000, A 0.000, B 0.000, C 0.000 }
gfCNCPoint2[14244] = {X 25.1126, Y 31.5019, Z -3.0000, A 0.000, B 0.000, C 0.000 }
gfCNCPoint2[14245] = {X 25.2522, Y 31.5424, Z -3.0000, A 0.000, B 0.000, C 0.000 }
gfCNCPoint2[14246] = {X 25.3902, Y 31.5877, Z -3.0000, A 0.000, B 0.000, C 0.000 }
gfCNCPoint2[14247] = {X 26.1378, Y 31.9316, Z -3.0000, A 0.000, B 0.000, C 0.000 }
gfCNCPoint2[14248] = {X 26.8048, Y 32.4134, Z -3.0000, A 0.000, B 0.000, C 0.000 }
gfCNCPoint2[14249] = {X 27.3662, Y 33.0149, Z -3.0000, A 0.000, B 0.000, C 0.000 }
gfCNCPoint2[14250] = {X 27.8009, Y 33.7136, Z -3.0000, A 0.000, B 0.000, C 0.000 }
gfCNCPoint2[14251] = {X 30.8380, Y 39.9879, Z -3.0000, A 0.000, B 0.000, C 0.000 }
gfCNCPoint2[14252] = {X 31.1526, Y 40.8802, Z -3.0000, A 0.000, B 0.000, C 0.000 }
gfCNCPoint2[14253] = {X 31.2615, Y 41.8200, Z -3.0000, A 0.000, B 0.000, C 0.000 }
gfCNCPoint2[14254] = {X 31.1593, Y 42.7606, Z -3.0000, A 0.000, B 0.000, C 0.000 }
gfCNCPoint2[14255] = {X 30.8511, Y 43.6551, Z -3.0000, A 0.000, B 0.000, C 0.000 }
gfCNCPoint2[14256] = {X 30.3522, Y 44.4590, Z -3.0000, A 0.000, B 0.000, C 0.000 }
gfCNCPoint2[14257] = {X 29.6874, Y 45.1323, Z -3.0000, A 0.000, B 0.000, C 0.000 }
gfCNCPoint2[14258] = {X 29.1512, Y 45.5658, Z -3.0000, A 0.000, B 0.000, C 0.000 }
gfCNCPoint2[14259] = {X 28.4535, Y 46.0236, Z -3.0000, A 0.000, B 0.000, C 0.000 }
gfCNCPoint2[14260] = {X 27.6799, Y 46.3365, Z -3.0000, A 0.000, B 0.000, C 0.000 }
gfCNCPoint2[14261] = {X 26.8602, Y 46.4925, Z -3.0000, A 0.000, B 0.000, C 0.000 }
gfCNCPoint2[14262] = {X 26.0257, Y 46.4855, Z -3.0000, A 0.000, B 0.000, C 0.000 }
gfCNCPoint2[14263] = {X 25.2087, Y 46.3158, Z -3.0000, A 0.000, B 0.000, C 0.000 }
gfCNCPoint2[14264] = {X 23.6269, Y 47.1651, Z -3.0000, A 0.000, B 0.000, C 0.000 }
gfCNCPoint2[14265] = {X 21.9938, Y 47.9108, Z -3.0000, A 0.000, B 0.000, C 0.000 }
gfCNCPoint2[14266] = {X 20.3161, Y 48.5500, Z -3.0000, A 0.000, B 0.000, C 0.000 }
gfCNCPoint2[14267] = {X 18.3979, Y 49.1581, Z -3.0000, A 0.000, B 0.000, C 0.000 }
gfCNCPoint2[14268] = {X 16.4334, Y 49.5942, Z -3.0000, A 0.000, B 0.000, C 0.000 }
gfCNCPoint2[14269] = {X 14.4380, Y 49.8549, Z -3.0000, A 0.000, B 0.000, C 0.000 }
gfCNCPoint2[14270] = {X 12.4274, Y 49.9381, Z -3.0000, A 0.000, B 0.000, C 0.000 }
gfCNCPoint2[14271] = {X 10.4173, Y 49.8433, Z -3.0000, A 0.000, B 0.000, C 0.000 }
gfCNCPoint2[14272] = {X 8.4235, Y 49.5712, Z -3.0000, A 0.000, B 0.000, C 0.000 }
gfCNCPoint2[14273] = {X 6.5546, Y 49.1376, Z -3.0000, A 0.000, B 0.000, C 0.000 }
gfCNCPoint2[14274] = {X 4.7463, Y 48.4969, Z -3.0000, A 0.000, B 0.000, C 0.000 }
gfCNCPoint2[14275] = {X 3.0212, Y 47.6573, Z -3.0000, A 0.000, B 0.000, C 0.000 }
gfCNCPoint2[14276] = {X 1.4014, Y 46.6292, Z -3.0000, A 0.000, B 0.000, C 0.000 }
gfCNCPoint2[14277] = {X 0.0840, Y 45.5688, Z -3.0000, A 0.000, B 0.000, C 0.000 }
gfCNCPoint2[14278] = {X -1.0871, Y 44.3487, Z -3.0000, A 0.000, B 0.000, C 0.000 }
gfCNCPoint2[14279] = {X -2.0927, Y 42.9890, Z -3.0000, A 0.000, B 0.000, C 0.000 }
gfCNCPoint2[14280] = {X -2.9164, Y 41.5119, Z -3.0000, A 0.000, B 0.000, C 0.000 }
gfCNCPoint2[14281] = {X -3.5445, Y 39.9417, Z -3.0000, A 0.000, B 0.000, C 0.000 }
gfCNCPoint2[14282] = {X -3.6229, Y 39.6938, Z -3.0000, A 0.000, B 0.000, C 0.000 }
gfCNCPoint2[14283] = {X -3.6965, Y 39.4444, Z -3.0000, A 0.000, B 0.000, C 0.000 }
gfCNCPoint2[14284] = {X -4.7907, Y 35.5970, Z -3.0000, A 0.000, B 0.000, C 0.000 }
gfCNCPoint2[14285] = {X -8.0020, Y 35.6621, Z -3.0000, A 0.000, B 0.000, C 0.000 }
gfCNCPoint2[14286] = {X -8.0020, Y 35.6621, Z 0.0000, A 0.000, B 0.000, C 0.000 }
gfCNCPoint2[14287] = {X -8.0020, Y 35.6621, Z 11.0000, A 0.000, B 0.000, C 0.000 }
gfCNCPoint2[14288] = {X -7.6965, Y 17.3009, Z 11.0000, A 0.000, B 0.000, C 0.000 }
gfCNCPoint2[14289] = {X -7.6965, Y 17.3009, Z 0.0000, A 0.000, B 0.000, C 0.000 }
gfCNCPoint2[14290] = {X -7.6965, Y 17.3009, Z -3.0000, A 0.000, B 0.000, C 0.000 }
gfCNCPoint2[14291] = {X -4.2194, Y 17.3009, Z -3.0000, A 0.000, B 0.000, C 0.000 }
gfCNCPoint2[14292] = {X -3.6965, Y 13.3353, Z -3.0000, A 0.000, B 0.000, C 0.000 }
gfCNCPoint2[14293] = {X -3.6095, Y 12.8762, Z -3.0000, A 0.000, B 0.000, C 0.000 }
gfCNCPoint2[14294] = {X -3.4716, Y 12.4297, Z -3.0000, A 0.000, B 0.000, C 0.000 }
gfCNCPoint2[14295] = {X -3.0335, Y 11.5715, Z -3.0000, A 0.000, B 0.000, C 0.000 }
gfCNCPoint2[14296] = {X -2.4097, Y 10.8370, Z -3.0000, A 0.000, B 0.000, C 0.000 }
gfCNCPoint2[14297] = {X -1.6337, Y 10.2658, Z -3.0000, A 0.000, B 0.000, C 0.000 }
gfCNCPoint2[14298] = {X -1.0364, Y 9.9251, Z -3.0000, A 0.000, B 0.000, C 0.000 }
gfCNCPoint2[14299] = {X -0.1656, Y 9.5524, Z -3.0000, A 0.000, B 0.000, C 0.000 }
gfCNCPoint2[14300] = {X 0.7669, Y 9.3865, Z -3.0000, A 0.000, B 0.000, C 0.000 }
gfCNCPoint2[14301] = {X 1.7128, Y 9.4357, Z -3.0000, A 0.000, B 0.000, C 0.000 }
gfCNCPoint2[14302] = {X 2.6231, Y 9.6977, Z -3.0000, A 0.000, B 0.000, C 0.000 }
gfCNCPoint2[14303] = {X 3.4232, Y 9.3195, Z -3.0000, A 0.000, B 0.000, C 0.000 }
gfCNCPoint2[14304] = {X 4.2470, Y 8.9962, Z -3.0000, A 0.000, B 0.000, C 0.000 }
gfCNCPoint2[14305] = {X 6.1462, Y 8.3307, Z -3.0000, A 0.000, B 0.000, C 0.000 }
gfCNCPoint2[14306] = {X 8.0957, Y 7.8316, Z -3.0000, A 0.000, B 0.000, C 0.000 }
gfCNCPoint2[14307] = {X 10.0810, Y 7.5026, Z -3.0000, A 0.000, B 0.000, C 0.000 }
gfCNCPoint2[14308] = {X 12.0874, Y 7.3462, Z -3.0000, A 0.000, B 0.000, C 0.000 }
gfCNCPoint2[14309] = {X 14.0997, Y 7.3636, Z -3.0000, A 0.000, B 0.000, C 0.000 }
gfCNCPoint2[14310] = {X 16.1030, Y 7.5547, Z -3.0000, A 0.000, B 0.000, C 0.000 }
gfCNCPoint2[14311] = {X 17.9097, Y 7.8852, Z -3.0000, A 0.000, B 0.000, C 0.000 }
gfCNCPoint2[14312] = {X 19.6711, Y 8.4054, Z -3.0000, A 0.000, B 0.000, C 0.000 }
gfCNCPoint2[14313] = {X 21.3675, Y 9.1095, Z -3.0000, A 0.000, B 0.000, C 0.000 }
gfCNCPoint2[14314] = {X 22.9796, Y 9.9895, Z -3.0000, A 0.000, B 0.000, C 0.000 }
gfCNCPoint2[14315] = {X 24.4894, Y 11.0355, Z -3.0000, A 0.000, B 0.000, C 0.000 }
gfCNCPoint2[14316] = {X 25.5611, Y 11.9725, Z -3.0000, A 0.000, B 0.000, C 0.000 }
gfCNCPoint2[14317] = {X 26.5224, Y 13.0224, Z -3.0000, A 0.000, B 0.000, C 0.000 }
gfCNCPoint2[14318] = {X 27.3615, Y 14.1724, Z -3.0000, A 0.000, B 0.000, C 0.000 }
gfCNCPoint2[14319] = {X 28.0681, Y 15.4082, Z -3.0000, A 0.000, B 0.000, C 0.000 }
gfCNCPoint2[14320] = {X 28.6334, Y 16.7147, Z -3.0000, A 0.000, B 0.000, C 0.000 }
gfCNCPoint2[14321] = {X 29.1026, Y 18.3529, Z -3.0000, A 0.000, B 0.000, C 0.000 }
gfCNCPoint2[14322] = {X 29.3810, Y 20.0340, Z -3.0000, A 0.000, B 0.000, C 0.000 }
gfCNCPoint2[14323] = {X 29.4649, Y 21.7360, Z -3.0000, A 0.000, B 0.000, C 0.000 }
gfCNCPoint2[14324] = {X 29.3533, Y 23.4364, Z -3.0000, A 0.000, B 0.000, C 0.000 }
gfCNCPoint2[14325] = {X 29.0476, Y 25.1129, Z -3.0000, A 0.000, B 0.000, C 0.000 }
gfCNCPoint2[14326] = {X 28.5894, Y 26.5979, Z -3.0000, A 0.000, B 0.000, C 0.000 }
gfCNCPoint2[14327] = {X 27.9356, Y 28.0077, Z -3.0000, A 0.000, B 0.000, C 0.000 }
gfCNCPoint2[14328] = {X 27.0982, Y 29.3169, Z -3.0000, A 0.000, B 0.000, C 0.000 }
gfCNCPoint2[14329] = {X 26.0922, Y 30.5015, Z -3.0000, A 0.000, B 0.000, C 0.000 }
gfCNCPoint2[14330] = {X 24.9361, Y 31.5400, Z -3.0000, A 0.000, B 0.000, C 0.000 }
gfCNCPoint2[14331] = {X 25.1517, Y 31.5959, Z -3.0000, A 0.000, B 0.000, C 0.000 }
gfCNCPoint2[14332] = {X 25.3640, Y 31.6633, Z -3.0000, A 0.000, B 0.000, C 0.000 }
gfCNCPoint2[14333] = {X 26.0974, Y 32.0007, Z -3.0000, A 0.000, B 0.000, C 0.000 }
gfCNCPoint2[14334] = {X 26.7519, Y 32.4734, Z -3.0000, A 0.000, B 0.000, C 0.000 }
gfCNCPoint2[14335] = {X 27.3027, Y 33.0636, Z -3.0000, A 0.000, B 0.000, C 0.000 }
gfCNCPoint2[14336] = {X 27.7292, Y 33.7491, Z -3.0000, A 0.000, B 0.000, C 0.000 }
gfCNCPoint2[14337] = {X 30.7660, Y 40.0227, Z -3.0000, A 0.000, B 0.000, C 0.000 }
gfCNCPoint2[14338] = {X 31.0747, Y 40.8982, Z -3.0000, A 0.000, B 0.000, C 0.000 }
gfCNCPoint2[14339] = {X 31.1815, Y 41.8203, Z -3.0000, A 0.000, B 0.000, C 0.000 }
gfCNCPoint2[14340] = {X 31.0813, Y 42.7431, Z -3.0000, A 0.000, B 0.000, C 0.000 }
gfCNCPoint2[14341] = {X 30.7789, Y 43.6208, Z -3.0000, A 0.000, B 0.000, C 0.000 }
gfCNCPoint2[14342] = {X 30.2893, Y 44.4095, Z -3.0000, A 0.000, B 0.000, C 0.000 }
gfCNCPoint2[14343] = {X 29.6371, Y 45.0700, Z -3.0000, A 0.000, B 0.000, C 0.000 }
gfCNCPoint2[14344] = {X 29.1010, Y 45.5036, Z -3.0000, A 0.000, B 0.000, C 0.000 }
gfCNCPoint2[14345] = {X 28.4102, Y 45.9560, Z -3.0000, A 0.000, B 0.000, C 0.000 }
gfCNCPoint2[14346] = {X 27.6439, Y 46.2637, Z -3.0000, A 0.000, B 0.000, C 0.000 }
gfCNCPoint2[14347] = {X 26.8320, Y 46.4146, Z -3.0000, A 0.000, B 0.000, C 0.000 }
gfCNCPoint2[14348] = {X 26.0064, Y 46.4029, Z -3.0000, A 0.000, B 0.000, C 0.000 }
gfCNCPoint2[14349] = {X 25.1991, Y 46.2289, Z -3.0000, A 0.000, B 0.000, C 0.000 }
gfCNCPoint2[14350] = {X 23.6122, Y 47.0830, Z -3.0000, A 0.000, B 0.000, C 0.000 }
gfCNCPoint2[14351] = {X 21.9733, Y 47.8327, Z -3.0000, A 0.000, B 0.000, C 0.000 }
gfCNCPoint2[14352] = {X 20.2893, Y 48.4746, Z -3.0000, A 0.000, B 0.000, C 0.000 }
gfCNCPoint2[14353] = {X 18.3777, Y 49.0806, Z -3.0000, A 0.000, B 0.000, C 0.000 }
gfCNCPoint2[14354] = {X 16.4199, Y 49.5153, Z -3.0000, A 0.000, B 0.000, C 0.000 }
gfCNCPoint2[14355] = {X 14.4314, Y 49.7751, Z -3.0000, A 0.000, B 0.000, C 0.000 }
gfCNCPoint2[14356] = {X 12.4277, Y 49.8581, Z -3.0000, A 0.000, B 0.000, C 0.000 }
gfCNCPoint2[14357] = {X 10.4245, Y 49.7637, Z -3.0000, A 0.000, B 0.000, C 0.000 }
gfCNCPoint2[14358] = {X 8.4375, Y 49.4924, Z -3.0000, A 0.000, B 0.000, C 0.000 }
gfCNCPoint2[14359] = {X 6.5772, Y 49.0609, Z -3.0000, A 0.000, B 0.000, C 0.000 }
gfCNCPoint2[14360] = {X 4.7772, Y 48.4231, Z -3.0000, A 0.000, B 0.000, C 0.000 }
gfCNCPoint2[14361] = {X 3.0601, Y 47.5873, Z -3.0000, A 0.000, B 0.000, C 0.000 }
gfCNCPoint2[14362] = {X 1.4477, Y 46.5640, Z -3.0000, A 0.000, B 0.000, C 0.000 }
gfCNCPoint2[14363] = {X 0.1382, Y 45.5100, Z -3.0000, A 0.000, B 0.000, C 0.000 }
gfCNCPoint2[14364] = {X -1.0259, Y 44.2973, Z -3.0000, A 0.000, B 0.000, C 0.000 }
gfCNCPoint2[14365] = {X -2.0254, Y 42.9457, Z -3.0000, A 0.000, B 0.000, C 0.000 }
gfCNCPoint2[14366] = {X -2.8441, Y 41.4775, Z -3.0000, A 0.000, B 0.000, C 0.000 }
gfCNCPoint2[14367] = {X -3.4684, Y 39.9168, Z -3.0000, A 0.000, B 0.000, C 0.000 }
gfCNCPoint2[14368] = {X -3.5885, Y 39.5302, Z -3.0000, A 0.000, B 0.000, C 0.000 }
gfCNCPoint2[14369] = {X -3.6965, Y 39.1400, Z -3.0000, A 0.000, B 0.000, C 0.000 }
gfCNCPoint2[14370] = {X -4.7046, Y 35.2691, Z -3.0000, A 0.000, B 0.000, C 0.000 }
gfCNCPoint2[14371] = {X -8.0057, Y 35.2638, Z -3.0000, A 0.000, B 0.000, C 0.000 }
gfCNCPoint2[14372] = {X -8.0057, Y 35.2638, Z 0.0000, A 0.000, B 0.000, C 0.000 }
gfCNCPoint2[14373] = {X -8.0057, Y 35.2638, Z 11.0000, A 0.000, B 0.000, C 0.000 }
gfCNCPoint2[14374] = {X -7.9994, Y 34.8111, Z 11.0000, A 0.000, B 0.000, C 0.000 }
gfCNCPoint2[14375] = {X -7.9994, Y 34.8111, Z 0.0000, A 0.000, B 0.000, C 0.000 }
gfCNCPoint2[14376] = {X -7.9994, Y 34.8111, Z -3.0000, A 0.000, B 0.000, C 0.000 }
gfCNCPoint2[14377] = {X -4.8620, Y 34.8943, Z -3.0000, A 0.000, B 0.000, C 0.000 }
gfCNCPoint2[14378] = {X -3.6965, Y 31.0679, Z -3.0000, A 0.000, B 0.000, C 0.000 }
gfCNCPoint2[14379] = {X -3.6590, Y 30.9466, Z -3.0000, A 0.000, B 0.000, C 0.000 }
gfCNCPoint2[14380] = {X -3.6204, Y 30.8257, Z -3.0000, A 0.000, B 0.000, C 0.000 }
gfCNCPoint2[14381] = {X -3.2922, Y 29.9167, Z -3.0000, A 0.000, B 0.000, C 0.000 }
gfCNCPoint2[14382] = {X -2.9041, Y 29.0315, Z -3.0000, A 0.000, B 0.000, C 0.000 }
gfCNCPoint2[14383] = {X -2.2644, Y 27.8853, Z -3.0000, A 0.000, B 0.000, C 0.000 }
gfCNCPoint2[14384] = {X -1.4893, Y 26.8259, Z -3.0000, A 0.000, B 0.000, C 0.000 }
gfCNCPoint2[14385] = {X -0.5905, Y 25.8693, Z -3.0000, A 0.000, B 0.000, C 0.000 }
gfCNCPoint2[14386] = {X 0.4186, Y 25.0297, Z -3.0000, A 0.000, B 0.000, C 0.000 }
gfCNCPoint2[14387] = {X 1.5227, Y 24.3199, Z -3.0000, A 0.000, B 0.000, C 0.000 }
gfCNCPoint2[14388] = {X 0.7349, Y 23.9289, Z -3.0000, A 0.000, B 0.000, C 0.000 }
gfCNCPoint2[14389] = {X 0.0425, Y 23.3865, Z -3.0000, A 0.000, B 0.000, C 0.000 }
gfCNCPoint2[14390] = {X -0.5256, Y 22.7152, Z -3.0000, A 0.000, B 0.000, C 0.000 }
gfCNCPoint2[14391] = {X -0.9460, Y 21.9427, Z -3.0000, A 0.000, B 0.000, C 0.000 }
gfCNCPoint2[14392] = {X -3.6215, Y 15.3843, Z -3.0000, A 0.000, B 0.000, C 0.000 }
gfCNCPoint2[14393] = {X -3.6605, Y 15.2750, Z -3.0000, A 0.000, B 0.000, C 0.000 }
gfCNCPoint2[14394] = {X -3.6965, Y 15.1646, Z -3.0000, A 0.000, B 0.000, C 0.000 }
gfCNCPoint2[14395] = {X -4.8868, Y 11.3458, Z -3.0000, A 0.000, B 0.000, C 0.000 }
gfCNCPoint2[14396] = {X -7.6965, Y 11.3458, Z -3.0000, A 0.000, B 0.000, C 0.000 }
gfCNCPoint2[14397] = {X -7.6965, Y 11.3458, Z 0.0000, A 0.000, B 0.000, C 0.000 }
gfCNCPoint2[14398] = {X -7.6965, Y 11.3458, Z 11.0000, A 0.000, B 0.000, C 0.000 }
gfCNCPoint2[14399] = {X -8.0054, Y 35.1786, Z 11.0000, A 0.000, B 0.000, C 0.000 }
gfCNCPoint2[14400] = {X -8.0054, Y 35.1786, Z 0.0000, A 0.000, B 0.000, C 0.000 }
gfCNCPoint2[14401] = {X -8.0054, Y 35.1786, Z -3.0000, A 0.000, B 0.000, C 0.000 }
gfCNCPoint2[14402] = {X -4.7899, Y 35.1989, Z -3.0000, A 0.000, B 0.000, C 0.000 }
gfCNCPoint2[14403] = {X -3.6965, Y 31.3512, Z -3.0000, A 0.000, B 0.000, C 0.000 }
gfCNCPoint2[14404] = {X -3.6227, Y 31.1001, Z -3.0000, A 0.000, B 0.000, C 0.000 }
gfCNCPoint2[14405] = {X -3.5443, Y 30.8503, Z -3.0000, A 0.000, B 0.000, C 0.000 }
gfCNCPoint2[14406] = {X -3.2179, Y 29.9463, Z -3.0000, A 0.000, B 0.000, C 0.000 }
gfCNCPoint2[14407] = {X -2.8320, Y 29.0660, Z -3.0000, A 0.000, B 0.000, C 0.000 }
gfCNCPoint2[14408] = {X -2.0401, Y 27.6909, Z -3.0000, A 0.000, B 0.000, C 0.000 }
gfCNCPoint2[14409] = {X -1.0524, Y 26.4488, Z -3.0000, A 0.000, B 0.000, C 0.000 }
gfCNCPoint2[14410] = {X 0.1092, Y 25.3676, Z -3.0000, A 0.000, B 0.000, C 0.000 }
gfCNCPoint2[14411] = {X 1.4187, Y 24.4712, Z -3.0000, A 0.000, B 0.000, C 0.000 }
gfCNCPoint2[14412] = {X 1.5678, Y 24.3863, Z -3.0000, A 0.000, B 0.000, C 0.000 }
gfCNCPoint2[14413] = {X 1.7183, Y 24.3038, Z -3.0000, A 0.000, B 0.000, C 0.000 }
gfCNCPoint2[14414] = {X 0.8913, Y 23.9305, Z -3.0000, A 0.000, B 0.000, C 0.000 }
gfCNCPoint2[14415] = {X 0.1626, Y 23.3898, Z -3.0000, A 0.000, B 0.000, C 0.000 }
gfCNCPoint2[14416] = {X -0.4343, Y 22.7065, Z -3.0000, A 0.000, B 0.000, C 0.000 }
gfCNCPoint2[14417] = {X -0.8722, Y 21.9118, Z -3.0000, A 0.000, B 0.000, C 0.000 }
gfCNCPoint2[14418] = {X -3.5465, Y 15.3564, Z -3.0000, A 0.000, B 0.000, C 0.000 }
gfCNCPoint2[14419] = {X -3.6290, Y 15.1119, Z -3.0000, A 0.000, B 0.000, C 0.000 }
gfCNCPoint2[14420] = {X -3.6965, Y 14.8629, Z -3.0000, A 0.000, B 0.000, C 0.000 }
gfCNCPoint2[14421] = {X -4.6246, Y 10.9720, Z -3.0000, A 0.000, B 0.000, C 0.000 }
gfCNCPoint2[14422] = {X -7.6965, Y 10.9720, Z -3.0000, A 0.000, B 0.000, C 0.000 }
gfCNCPoint2[14423] = {X -7.6965, Y 10.9720, Z 0.0000, A 0.000, B 0.000, C 0.000 }
gfCNCPoint2[14424] = {X -7.6965, Y 10.9720, Z 11.0000, A 0.000, B 0.000, C 0.000 }
gfCNCPoint2[14425] = {X -8.0036, Y 35.5748, Z 11.0000, A 0.000, B 0.000, C 0.000 }
gfCNCPoint2[14426] = {X -8.0036, Y 35.5748, Z 0.0000, A 0.000, B 0.000, C 0.000 }
gfCNCPoint2[14427] = {X -8.0036, Y 35.5748, Z -3.0000, A 0.000, B 0.000, C 0.000 }
gfCNCPoint2[14428] = {X -4.7114, Y 35.5239, Z -3.0000, A 0.000, B 0.000, C 0.000 }
gfCNCPoint2[14429] = {X -3.6965, Y 31.6547, Z -3.0000, A 0.000, B 0.000, C 0.000 }
gfCNCPoint2[14430] = {X -3.5879, Y 31.2632, Z -3.0000, A 0.000, B 0.000, C 0.000 }
gfCNCPoint2[14431] = {X -3.4682, Y 30.8750, Z -3.0000, A 0.000, B 0.000, C 0.000 }
gfCNCPoint2[14432] = {X -3.1436, Y 29.9760, Z -3.0000, A 0.000, B 0.000, C 0.000 }
gfCNCPoint2[14433] = {X -2.7598, Y 29.1006, Z -3.0000, A 0.000, B 0.000, C 0.000 }
gfCNCPoint2[14434] = {X -1.9739, Y 27.7358, Z -3.0000, A 0.000, B 0.000, C 0.000 }
gfCNCPoint2[14435] = {X -0.9936, Y 26.5031, Z -3.0000, A 0.000, B 0.000, C 0.000 }
gfCNCPoint2[14436] = {X 0.1592, Y 25.4300, Z -3.0000, A 0.000, B 0.000, C 0.000 }
gfCNCPoint2[14437] = {X 1.4588, Y 24.5404, Z -3.0000, A 0.000, B 0.000, C 0.000 }
gfCNCPoint2[14438] = {X 1.6920, Y 24.4091, Z -3.0000, A 0.000, B 0.000, C 0.000 }
gfCNCPoint2[14439] = {X 1.9284, Y 24.2837, Z -3.0000, A 0.000, B 0.000, C 0.000 }
gfCNCPoint2[14440] = {X 1.0582, Y 23.9328, Z -3.0000, A 0.000, B 0.000, C 0.000 }
gfCNCPoint2[14441] = {X 0.2887, Y 23.3958, Z -3.0000, A 0.000, B 0.000, C 0.000 }
gfCNCPoint2[14442] = {X -0.3408, Y 22.7001, Z -3.0000, A 0.000, B 0.000, C 0.000 }
gfCNCPoint2[14443] = {X -0.7984, Y 21.8809, Z -3.0000, A 0.000, B 0.000, C 0.000 }
gfCNCPoint2[14444] = {X -3.4716, Y 15.3285, Z -3.0000, A 0.000, B 0.000, C 0.000 }
